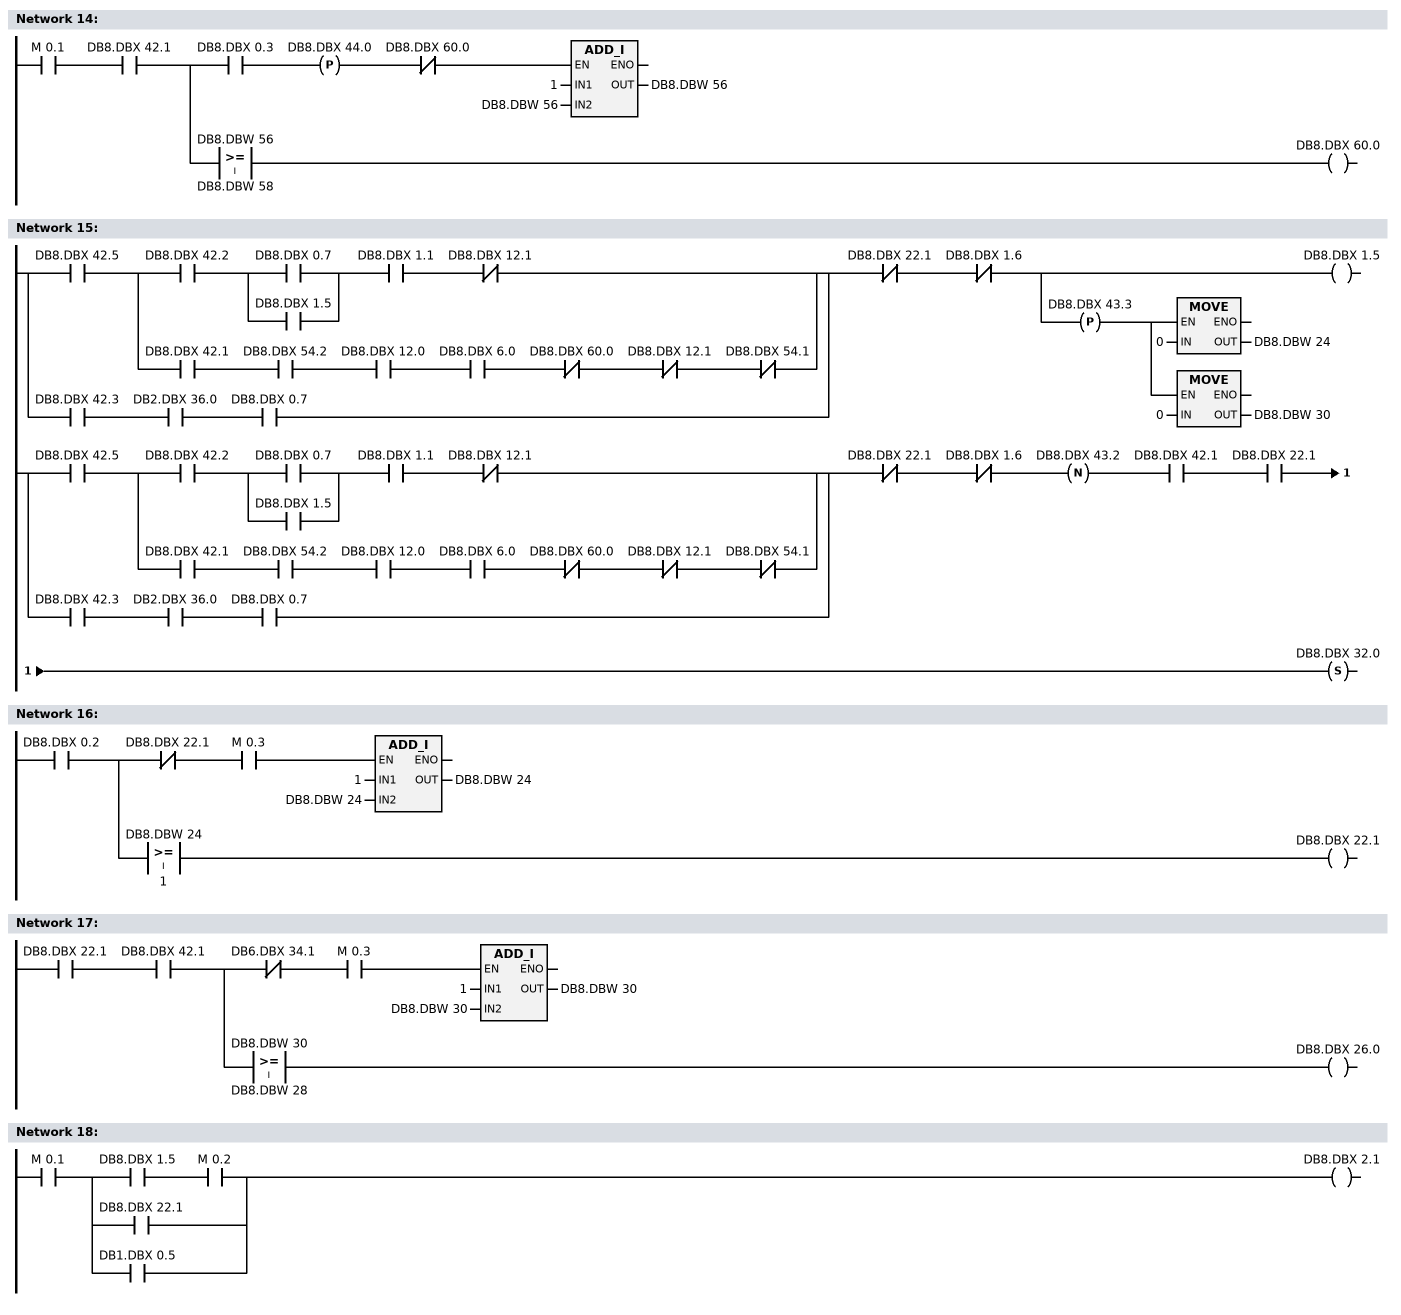
NETWORK
TITLE =
      A     M 0.1;
      A     DB8.DBX 42.1;
      =     L 0.0;
      A     L 0.0;
      A     DB8.DBX 0.3;
      FP    DB8.DBX 44.0;
      AN    DB8.DBX 60.0;
      JNB   M010;
      L     1;
      L     DB8.DBW 56;
      +I;
      T     DB8.DBW 56;
M010: NOP   0;
      A     L 0.0;
      A(;
      L     DB8.DBW 56;
      L     DB8.DBW 58;
      >=I;
      );
      =     DB8.DBX 60.0;
NETWORK
TITLE =
      A(;
      A     DB8.DBX 42.5;
      A(;
      A     DB8.DBX 42.2;
      A(;
      O     DB8.DBX 0.7;
      O     DB8.DBX 1.5;
      );
      A     DB8.DBX 1.1;
      AN    DB8.DBX 12.1;
      O;
      A     DB8.DBX 42.1;
      A     DB8.DBX 54.2;
      A     DB8.DBX 12.0;
      A     DB8.DBX 6.0;
      AN    DB8.DBX 60.0;
      AN    DB8.DBX 12.1;
      AN    DB8.DBX 54.1;
      );
      O;
      A     DB8.DBX 42.3;
      A     DB2.DBX 36.0;
      A     DB8.DBX 0.7;
      );
      AN    DB8.DBX 22.1;
      AN    DB8.DBX 1.6;
      =     L 0.0;
      A     L 0.0;
      BLD   102;
      =     DB8.DBX 1.5;
      A(;
      A     L 0.0;
      FN    DB8.DBX 43.2;
      );
      A     DB8.DBX 42.1;
      A     DB8.DBX 22.1;
      S     DB8.DBX 32.0;
      A     L 0.0;
      FP    DB8.DBX 43.3;
      =     L 0.1;
      A     L 0.1;
      JNB   M011;
      L     0;
      T     DB8.DBW 24;
M011: NOP   0;
      A     L 0.1;
      JNB   M012;
      L     0;
      T     DB8.DBW 30;
M012: NOP   0;
NETWORK
TITLE =
      A     DB8.DBX 0.2;
      =     L 0.0;
      A     L 0.0;
      AN    DB8.DBX 22.1;
      A     M 0.3;
      JNB   M013;
      L     1;
      L     DB8.DBW 24;
      +I;
      T     DB8.DBW 24;
M013: NOP   0;
      A     L 0.0;
      A(;
      L     DB8.DBW 24;
      L     1;
      >=I;
      );
      =     DB8.DBX 22.1;
NETWORK
TITLE =
      A     DB8.DBX 22.1;
      A     DB8.DBX 42.1;
      =     L 0.0;
      A     L 0.0;
      AN    DB6.DBX 34.1;
      A     M 0.3;
      JNB   M014;
      L     1;
      L     DB8.DBW 30;
      +I;
      T     DB8.DBW 30;
M014: NOP   0;
      A     L 0.0;
      A(;
      L     DB8.DBW 30;
      L     DB8.DBW 28;
      >=I;
      );
      =     DB8.DBX 26.0;
NETWORK
TITLE =
      A     M 0.1;
      A(;
      A     DB8.DBX 1.5;
      A     M 0.2;
      O     DB8.DBX 22.1;
      O     DB1.DBX 0.5;
      );
      =     DB8.DBX 2.1;
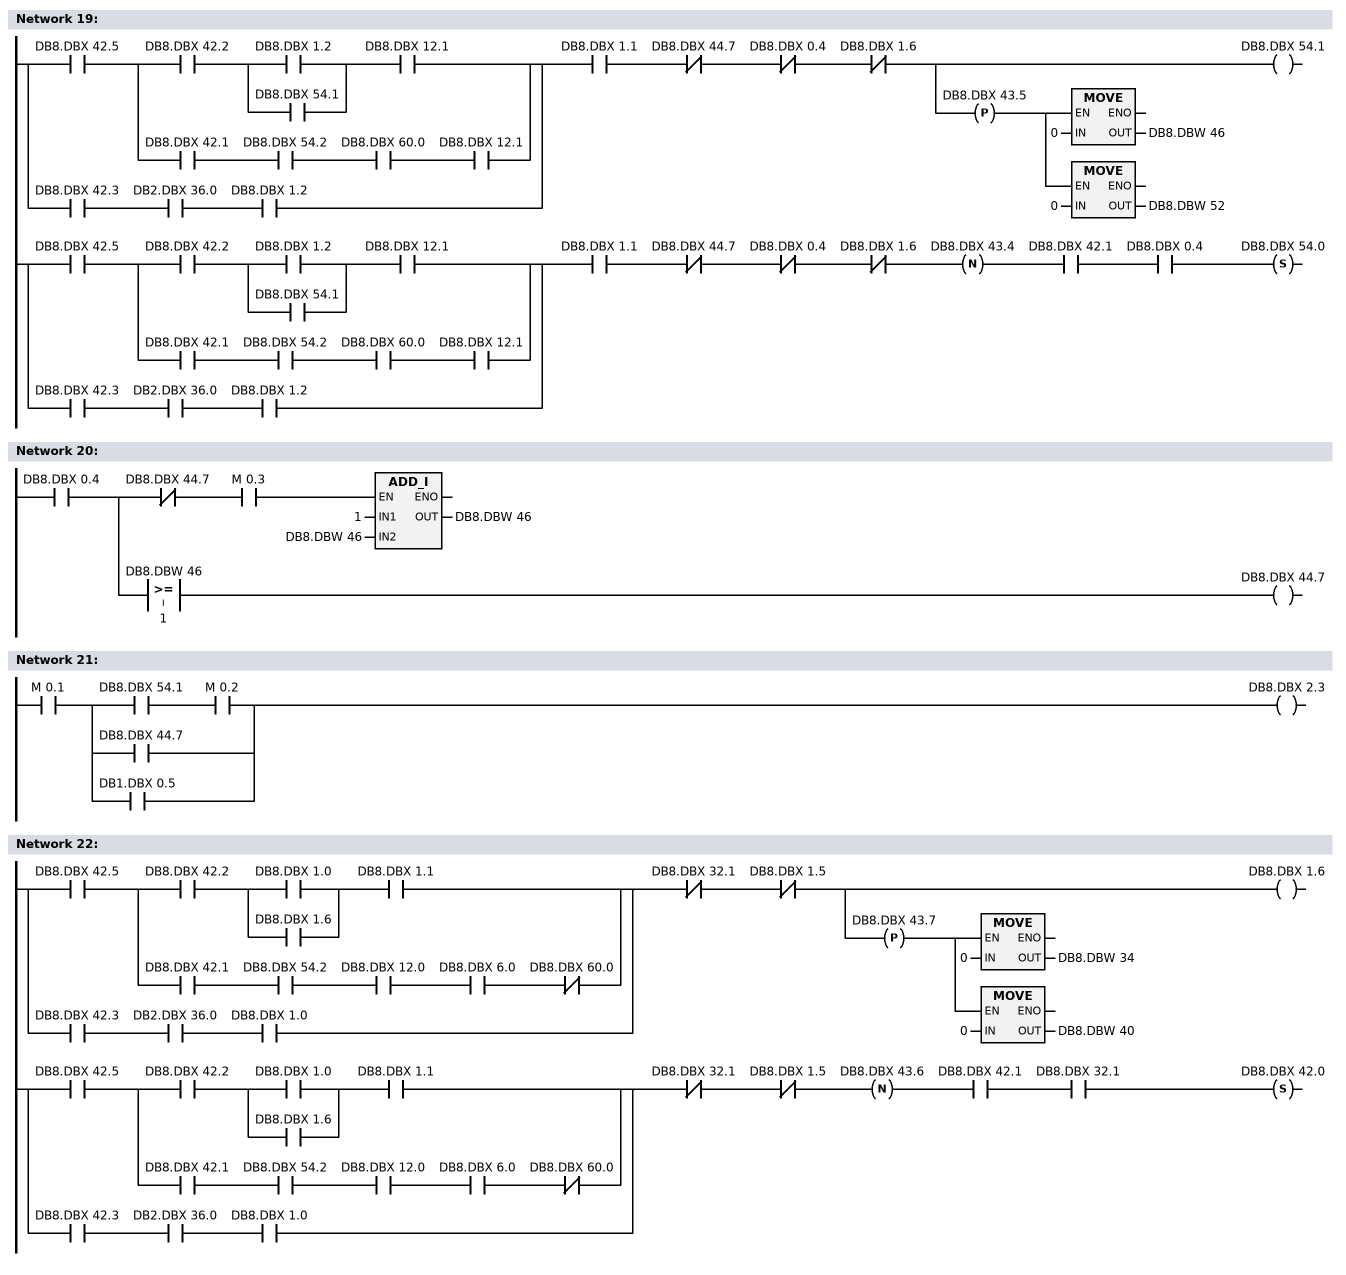
NETWORK
TITLE =
      A(;
      A     DB8.DBX 42.5;
      A(;
      A     DB8.DBX 42.2;
      A(;
      O     DB8.DBX 1.2;
      O     DB8.DBX 54.1;
      );
      A     DB8.DBX 12.1;
      O;
      A     DB8.DBX 42.1;
      A     DB8.DBX 54.2;
      A     DB8.DBX 60.0;
      A     DB8.DBX 12.1;
      );
      O;
      A     DB8.DBX 42.3;
      A     DB2.DBX 36.0;
      A     DB8.DBX 1.2;
      );
      A     DB8.DBX 1.1;
      AN    DB8.DBX 44.7;
      AN    DB8.DBX 0.4;
      AN    DB8.DBX 1.6;
      =     L 0.0;
      A     L 0.0;
      BLD   102;
      =     DB8.DBX 54.1;
      A(;
      A     L 0.0;
      FN    DB8.DBX 43.4;
      );
      A     DB8.DBX 42.1;
      A     DB8.DBX 0.4;
      S     DB8.DBX 54.0;
      A     L 0.0;
      FP    DB8.DBX 43.5;
      =     L 0.1;
      A     L 0.1;
      JNB   M015;
      L     0;
      T     DB8.DBW 46;
M015: NOP   0;
      A     L 0.1;
      JNB   M016;
      L     0;
      T     DB8.DBW 52;
M016: NOP   0;
NETWORK
TITLE =
      A     DB8.DBX 0.4;
      =     L 0.0;
      A     L 0.0;
      AN    DB8.DBX 44.7;
      A     M 0.3;
      JNB   M017;
      L     1;
      L     DB8.DBW 46;
      +I;
      T     DB8.DBW 46;
M017: NOP   0;
      A     L 0.0;
      A(;
      L     DB8.DBW 46;
      L     1;
      >=I;
      );
      =     DB8.DBX 44.7;
NETWORK
TITLE =
      A     M 0.1;
      A(;
      A     DB8.DBX 54.1;
      A     M 0.2;
      O     DB8.DBX 44.7;
      O     DB1.DBX 0.5;
      );
      =     DB8.DBX 2.3;
NETWORK
TITLE =
      A(;
      A     DB8.DBX 42.5;
      A(;
      A     DB8.DBX 42.2;
      A(;
      O     DB8.DBX 1.0;
      O     DB8.DBX 1.6;
      );
      A     DB8.DBX 1.1;
      O;
      A     DB8.DBX 42.1;
      A     DB8.DBX 54.2;
      A     DB8.DBX 12.0;
      A     DB8.DBX 6.0;
      AN    DB8.DBX 60.0;
      );
      O;
      A     DB8.DBX 42.3;
      A     DB2.DBX 36.0;
      A     DB8.DBX 1.0;
      );
      AN    DB8.DBX 32.1;
      AN    DB8.DBX 1.5;
      =     L 0.0;
      A     L 0.0;
      BLD   102;
      =     DB8.DBX 1.6;
      A(;
      A     L 0.0;
      FN    DB8.DBX 43.6;
      );
      A     DB8.DBX 42.1;
      A     DB8.DBX 32.1;
      S     DB8.DBX 42.0;
      A     L 0.0;
      FP    DB8.DBX 43.7;
      =     L 0.1;
      A     L 0.1;
      JNB   M018;
      L     0;
      T     DB8.DBW 34;
M018: NOP   0;
      A     L 0.1;
      JNB   M019;
      L     0;
      T     DB8.DBW 40;
M019: NOP   0;
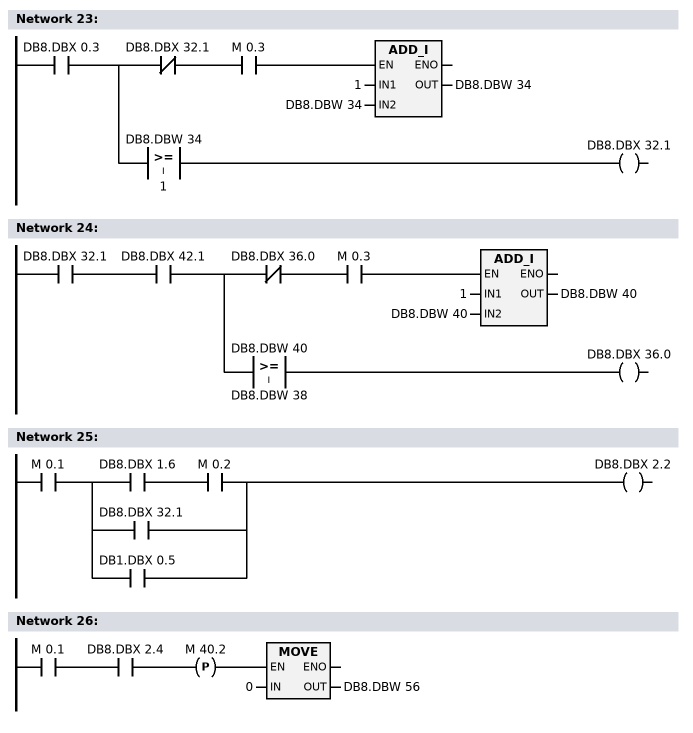
NETWORK
TITLE =
      A     DB8.DBX 0.3;
      =     L 0.0;
      A     L 0.0;
      AN    DB8.DBX 32.1;
      A     M 0.3;
      JNB   M020;
      L     1;
      L     DB8.DBW 34;
      +I;
      T     DB8.DBW 34;
M020: NOP   0;
      A     L 0.0;
      A(;
      L     DB8.DBW 34;
      L     1;
      >=I;
      );
      =     DB8.DBX 32.1;
NETWORK
TITLE =
      A     DB8.DBX 32.1;
      A     DB8.DBX 42.1;
      =     L 0.0;
      A     L 0.0;
      AN    DB8.DBX 36.0;
      A     M 0.3;
      JNB   M021;
      L     1;
      L     DB8.DBW 40;
      +I;
      T     DB8.DBW 40;
M021: NOP   0;
      A     L 0.0;
      A(;
      L     DB8.DBW 40;
      L     DB8.DBW 38;
      >=I;
      );
      =     DB8.DBX 36.0;
NETWORK
TITLE =
      A     M 0.1;
      A(;
      A     DB8.DBX 1.6;
      A     M 0.2;
      O     DB8.DBX 32.1;
      O     DB1.DBX 0.5;
      );
      =     DB8.DBX 2.2;
NETWORK
TITLE =
      A     M 0.1;
      A     DB8.DBX 2.4;
      FP    M 40.2;
      JNB   M022;
      L     0;
      T     DB8.DBW 56;
M022: NOP   0;
END_FUNCTION

FUNCTION FC 11 : VOID
AUTHOR : Kamillas
VERSION : 0.1
BEGIN
// (block stored without names or comments; labels and parameter names are numbered)
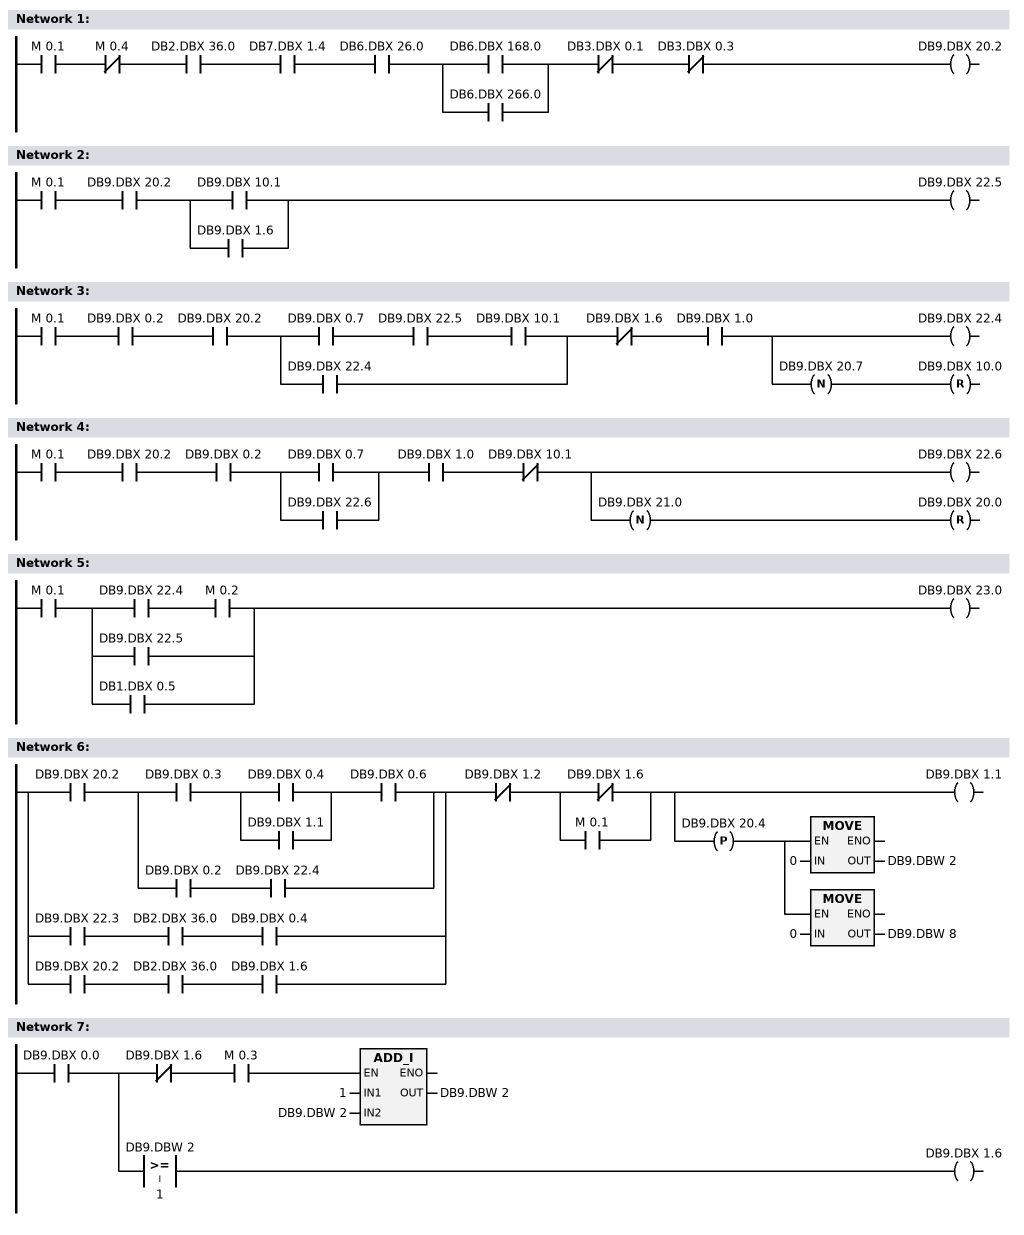
NETWORK
TITLE =
      A     M 0.1;
      AN    M 0.4;
      A     DB2.DBX 36.0;
      A     DB7.DBX 1.4;
      A     DB6.DBX 26.0;
      A(;
      O     DB6.DBX 168.0;
      O     DB6.DBX 266.0;
      );
      AN    DB3.DBX 0.1;
      AN    DB3.DBX 0.3;
      =     DB9.DBX 20.2;
NETWORK
TITLE =
      A     M 0.1;
      A     DB9.DBX 20.2;
      A(;
      O     DB9.DBX 10.1;
      O     DB9.DBX 1.6;
      );
      =     DB9.DBX 22.5;
NETWORK
TITLE =
      A     M 0.1;
      A     DB9.DBX 0.2;
      A     DB9.DBX 20.2;
      A(;
      A     DB9.DBX 0.7;
      A     DB9.DBX 22.5;
      A     DB9.DBX 10.1;
      O     DB9.DBX 22.4;
      );
      AN    DB9.DBX 1.6;
      A     DB9.DBX 1.0;
      =     L 0.0;
      A     L 0.0;
      BLD   102;
      =     DB9.DBX 22.4;
      A     L 0.0;
      FN    DB9.DBX 20.7;
      R     DB9.DBX 10.0;
NETWORK
TITLE =
      A     M 0.1;
      A     DB9.DBX 20.2;
      A     DB9.DBX 0.2;
      A(;
      O     DB9.DBX 0.7;
      O     DB9.DBX 22.6;
      );
      A     DB9.DBX 1.0;
      AN    DB9.DBX 10.1;
      =     L 0.0;
      A     L 0.0;
      BLD   102;
      =     DB9.DBX 22.6;
      A     L 0.0;
      FN    DB9.DBX 21.0;
      R     DB9.DBX 20.0;
NETWORK
TITLE =
      A     M 0.1;
      A(;
      A     DB9.DBX 22.4;
      A     M 0.2;
      O     DB9.DBX 22.5;
      O     DB1.DBX 0.5;
      );
      =     DB9.DBX 23.0;
NETWORK
TITLE =
      A(;
      A     DB9.DBX 20.2;
      A(;
      A     DB9.DBX 0.3;
      A(;
      O     DB9.DBX 0.4;
      O     DB9.DBX 1.1;
      );
      A     DB9.DBX 0.6;
      O;
      A     DB9.DBX 0.2;
      A     DB9.DBX 22.4;
      );
      O;
      A     DB9.DBX 22.3;
      A     DB2.DBX 36.0;
      A     DB9.DBX 0.4;
      O;
      A     DB9.DBX 20.2;
      A     DB2.DBX 36.0;
      A     DB9.DBX 1.6;
      );
      AN    DB9.DBX 1.2;
      A(;
      ON    DB9.DBX 1.6;
      O     M 0.1;
      );
      =     L 0.0;
      A     L 0.0;
      BLD   102;
      =     DB9.DBX 1.1;
      A     L 0.0;
      FP    DB9.DBX 20.4;
      =     L 0.1;
      A     L 0.1;
      JNB   M001;
      L     0;
      T     DB9.DBW 2;
M001: NOP   0;
      A     L 0.1;
      JNB   M002;
      L     0;
      T     DB9.DBW 8;
M002: NOP   0;
NETWORK
TITLE =
      A     DB9.DBX 0.0;
      =     L 0.0;
      A     L 0.0;
      AN    DB9.DBX 1.6;
      A     M 0.3;
      JNB   M003;
      L     1;
      L     DB9.DBW 2;
      +I;
      T     DB9.DBW 2;
M003: NOP   0;
      A     L 0.0;
      A(;
      L     DB9.DBW 2;
      L     1;
      >=I;
      );
      =     DB9.DBX 1.6;
NETWORK
TITLE =
      A     DB9.DBX 1.6;
      =     L 0.0;
      A     L 0.0;
      A     DB9.DBX 0.2;
      AN    DB9.DBX 4.0;
      A     M 0.3;
      JNB   M004;
      L     1;
      L     DB9.DBW 8;
      +I;
      T     DB9.DBW 8;
M004: NOP   0;
      A     L 0.0;
      A(;
      L     DB9.DBW 8;
      L     DB9.DBW 6;
      >=I;
      );
      =     L 0.1;
      A     L 0.1;
      A     DB9.DBX 0.2;
      =     DB9.DBX 4.0;
      A(;
      A     L 0.1;
      FP    DB9.DBX 20.3;
      );
      A     DB9.DBX 0.2;
      A     DB9.DBX 1.6;
      S     DB9.DBX 10.0;
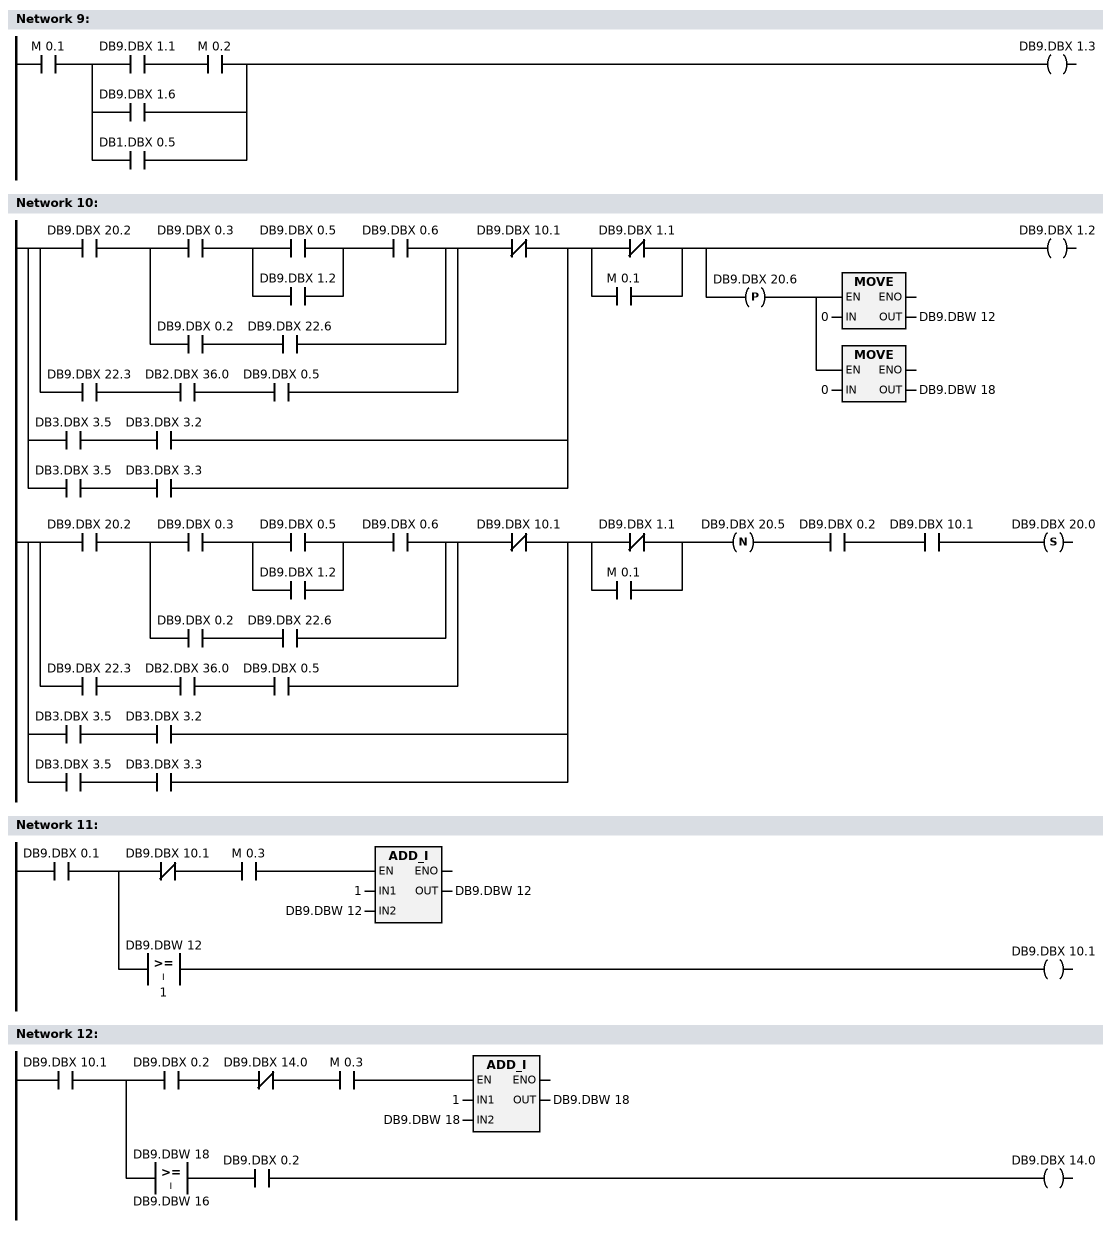
NETWORK
TITLE =
      A     M 0.1;
      A(;
      A     DB9.DBX 1.1;
      A     M 0.2;
      O     DB9.DBX 1.6;
      O     DB1.DBX 0.5;
      );
      =     DB9.DBX 1.3;
NETWORK
TITLE =
      A(;
      A(;
      A     DB9.DBX 20.2;
      A(;
      A     DB9.DBX 0.3;
      A(;
      O     DB9.DBX 0.5;
      O     DB9.DBX 1.2;
      );
      A     DB9.DBX 0.6;
      O;
      A     DB9.DBX 0.2;
      A     DB9.DBX 22.6;
      );
      O;
      A     DB9.DBX 22.3;
      A     DB2.DBX 36.0;
      A     DB9.DBX 0.5;
      );
      AN    DB9.DBX 10.1;
      O;
      A     DB3.DBX 3.5;
      A     DB3.DBX 3.2;
      O;
      A     DB3.DBX 3.5;
      A     DB3.DBX 3.3;
      );
      A(;
      ON    DB9.DBX 1.1;
      O     M 0.1;
      );
      =     L 0.0;
      A     L 0.0;
      BLD   102;
      =     DB9.DBX 1.2;
      A(;
      A     L 0.0;
      FN    DB9.DBX 20.5;
      );
      A     DB9.DBX 0.2;
      A     DB9.DBX 10.1;
      S     DB9.DBX 20.0;
      A     L 0.0;
      FP    DB9.DBX 20.6;
      =     L 0.1;
      A     L 0.1;
      JNB   M005;
      L     0;
      T     DB9.DBW 12;
M005: NOP   0;
      A     L 0.1;
      JNB   M006;
      L     0;
      T     DB9.DBW 18;
M006: NOP   0;
NETWORK
TITLE =
      A     DB9.DBX 0.1;
      =     L 0.0;
      A     L 0.0;
      AN    DB9.DBX 10.1;
      A     M 0.3;
      JNB   M007;
      L     1;
      L     DB9.DBW 12;
      +I;
      T     DB9.DBW 12;
M007: NOP   0;
      A     L 0.0;
      A(;
      L     DB9.DBW 12;
      L     1;
      >=I;
      );
      =     DB9.DBX 10.1;
NETWORK
TITLE =
      A     DB9.DBX 10.1;
      =     L 0.0;
      A     L 0.0;
      A     DB9.DBX 0.2;
      AN    DB9.DBX 14.0;
      A     M 0.3;
      JNB   M008;
      L     1;
      L     DB9.DBW 18;
      +I;
      T     DB9.DBW 18;
M008: NOP   0;
      A     L 0.0;
      A(;
      L     DB9.DBW 18;
      L     DB9.DBW 16;
      >=I;
      );
      A     DB9.DBX 0.2;
      =     DB9.DBX 14.0;
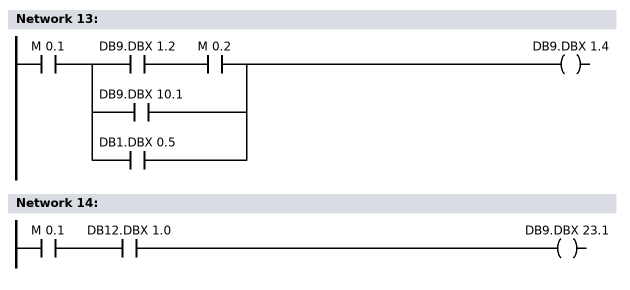
NETWORK
TITLE =
      A     M 0.1;
      A(;
      A     DB9.DBX 1.2;
      A     M 0.2;
      O     DB9.DBX 10.1;
      O     DB1.DBX 0.5;
      );
      =     DB9.DBX 1.4;
NETWORK
TITLE =
      A     M 0.1;
      A     DB12.DBX 1.0;
      =     DB9.DBX 23.1;
END_FUNCTION

FUNCTION FC 12 : VOID
AUTHOR : Kamillas
VERSION : 0.1
BEGIN
// (block stored without names or comments; labels and parameter names are numbered)
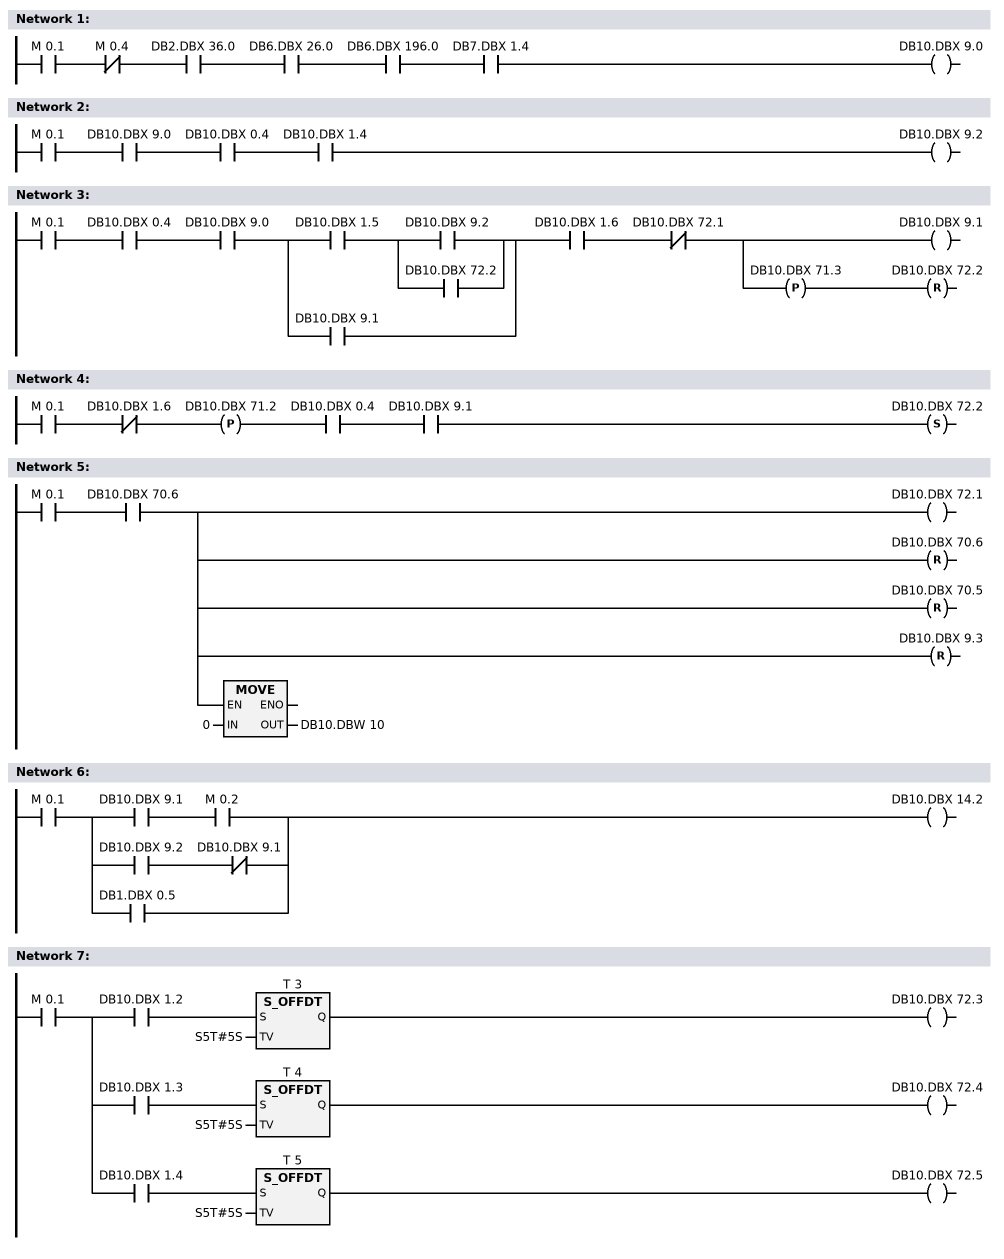
NETWORK
TITLE =
      A     M 0.1;
      AN    M 0.4;
      A     DB2.DBX 36.0;
      A     DB6.DBX 26.0;
      A     DB6.DBX 196.0;
      A     DB7.DBX 1.4;
      =     DB10.DBX 9.0;
NETWORK
TITLE =
      A     M 0.1;
      A     DB10.DBX 9.0;
      A     DB10.DBX 0.4;
      A     DB10.DBX 1.4;
      =     DB10.DBX 9.2;
NETWORK
TITLE =
      A     M 0.1;
      A     DB10.DBX 0.4;
      A     DB10.DBX 9.0;
      A(;
      A     DB10.DBX 1.5;
      A(;
      O     DB10.DBX 9.2;
      O     DB10.DBX 72.2;
      );
      O     DB10.DBX 9.1;
      );
      A     DB10.DBX 1.6;
      AN    DB10.DBX 72.1;
      =     L 0.0;
      A     L 0.0;
      BLD   102;
      =     DB10.DBX 9.1;
      A     L 0.0;
      FP    DB10.DBX 71.3;
      R     DB10.DBX 72.2;
NETWORK
TITLE =
      A     M 0.1;
      AN    DB10.DBX 1.6;
      FP    DB10.DBX 71.2;
      A     DB10.DBX 0.4;
      A     DB10.DBX 9.1;
      S     DB10.DBX 72.2;
NETWORK
TITLE =
      A     M 0.1;
      A     DB10.DBX 70.6;
      =     L 0.0;
      A     L 0.0;
      BLD   102;
      =     DB10.DBX 72.1;
      A     L 0.0;
      BLD   102;
      R     DB10.DBX 70.6;
      A     L 0.0;
      BLD   102;
      R     DB10.DBX 70.5;
      A     L 0.0;
      BLD   102;
      R     DB10.DBX 9.3;
      A     L 0.0;
      JNB   M001;
      L     0;
      T     DB10.DBW 10;
M001: NOP   0;
NETWORK
TITLE =
      A     M 0.1;
      A(;
      A     DB10.DBX 9.1;
      A     M 0.2;
      O;
      A     DB10.DBX 9.2;
      AN    DB10.DBX 9.1;
      O     DB1.DBX 0.5;
      );
      =     DB10.DBX 14.2;
NETWORK
TITLE =
      A     M 0.1;
      =     L 0.0;
      A     L 0.0;
      A     DB10.DBX 1.2;
      L     S5T#5S;
      SF    T 3;
      NOP   0;
      NOP   0;
      NOP   0;
      A     T 3;
      =     DB10.DBX 72.3;
      A     L 0.0;
      A     DB10.DBX 1.3;
      L     S5T#5S;
      SF    T 4;
      NOP   0;
      NOP   0;
      NOP   0;
      A     T 4;
      =     DB10.DBX 72.4;
      A     L 0.0;
      A     DB10.DBX 1.4;
      L     S5T#5S;
      SF    T 5;
      NOP   0;
      NOP   0;
      NOP   0;
      A     T 5;
      =     DB10.DBX 72.5;
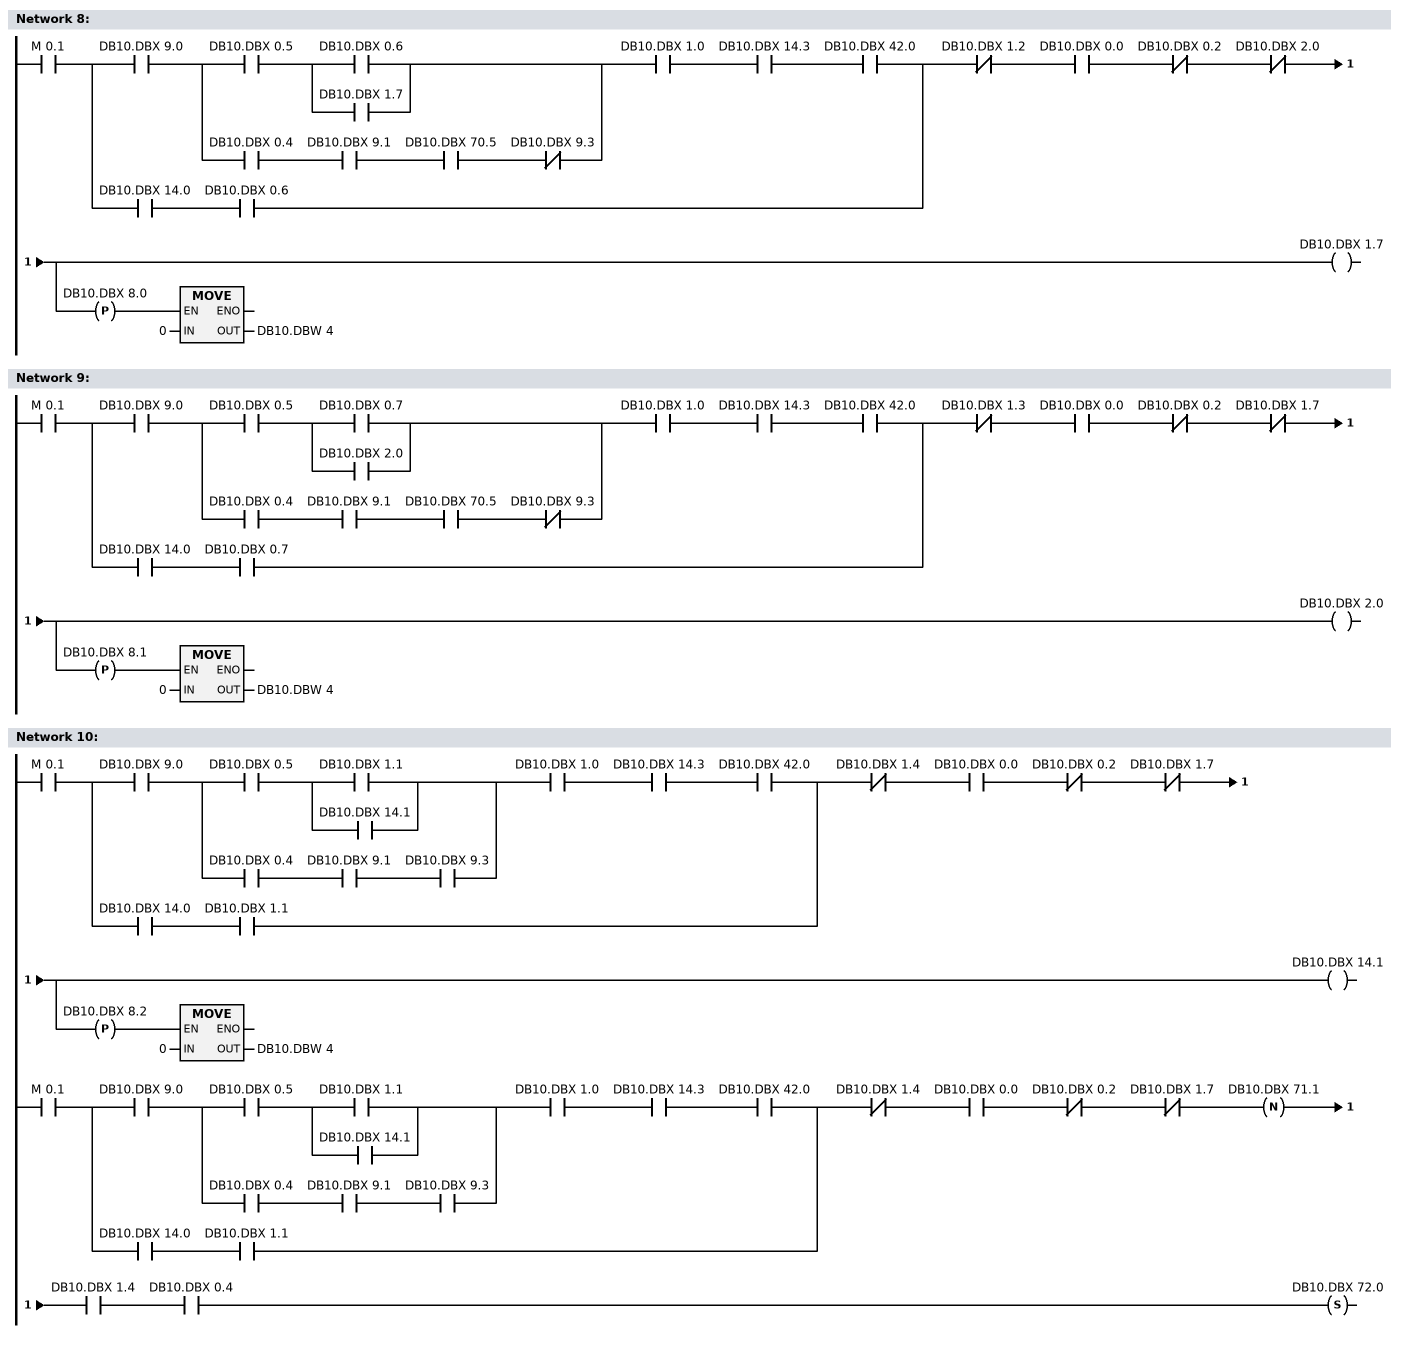
NETWORK
TITLE =
      A     M 0.1;
      A(;
      A     DB10.DBX 9.0;
      A(;
      A     DB10.DBX 0.5;
      A(;
      O     DB10.DBX 0.6;
      O     DB10.DBX 1.7;
      );
      O;
      A     DB10.DBX 0.4;
      A     DB10.DBX 9.1;
      A     DB10.DBX 70.5;
      AN    DB10.DBX 9.3;
      );
      A     DB10.DBX 1.0;
      A     DB10.DBX 14.3;
      A     DB10.DBX 42.0;
      O;
      A     DB10.DBX 14.0;
      A     DB10.DBX 0.6;
      );
      AN    DB10.DBX 1.2;
      A     DB10.DBX 0.0;
      AN    DB10.DBX 0.2;
      AN    DB10.DBX 2.0;
      =     L 0.0;
      A     L 0.0;
      BLD   102;
      =     DB10.DBX 1.7;
      A     L 0.0;
      FP    DB10.DBX 8.0;
      JNB   M002;
      L     0;
      T     DB10.DBW 4;
M002: NOP   0;
NETWORK
TITLE =
      A     M 0.1;
      A(;
      A     DB10.DBX 9.0;
      A(;
      A     DB10.DBX 0.5;
      A(;
      O     DB10.DBX 0.7;
      O     DB10.DBX 2.0;
      );
      O;
      A     DB10.DBX 0.4;
      A     DB10.DBX 9.1;
      A     DB10.DBX 70.5;
      AN    DB10.DBX 9.3;
      );
      A     DB10.DBX 1.0;
      A     DB10.DBX 14.3;
      A     DB10.DBX 42.0;
      O;
      A     DB10.DBX 14.0;
      A     DB10.DBX 0.7;
      );
      AN    DB10.DBX 1.3;
      A     DB10.DBX 0.0;
      AN    DB10.DBX 0.2;
      AN    DB10.DBX 1.7;
      =     L 0.0;
      A     L 0.0;
      BLD   102;
      =     DB10.DBX 2.0;
      A     L 0.0;
      FP    DB10.DBX 8.1;
      JNB   M003;
      L     0;
      T     DB10.DBW 4;
M003: NOP   0;
NETWORK
TITLE =
      A     M 0.1;
      A(;
      A     DB10.DBX 9.0;
      A(;
      A     DB10.DBX 0.5;
      A(;
      O     DB10.DBX 1.1;
      O     DB10.DBX 14.1;
      );
      O;
      A     DB10.DBX 0.4;
      A     DB10.DBX 9.1;
      A     DB10.DBX 9.3;
      );
      A     DB10.DBX 1.0;
      A     DB10.DBX 14.3;
      A     DB10.DBX 42.0;
      O;
      A     DB10.DBX 14.0;
      A     DB10.DBX 1.1;
      );
      AN    DB10.DBX 1.4;
      A     DB10.DBX 0.0;
      AN    DB10.DBX 0.2;
      AN    DB10.DBX 1.7;
      =     L 0.0;
      A     L 0.0;
      BLD   102;
      =     DB10.DBX 14.1;
      A(;
      A     L 0.0;
      FN    DB10.DBX 71.1;
      );
      A     DB10.DBX 1.4;
      A     DB10.DBX 0.4;
      S     DB10.DBX 72.0;
      A     L 0.0;
      FP    DB10.DBX 8.2;
      JNB   M004;
      L     0;
      T     DB10.DBW 4;
M004: NOP   0;
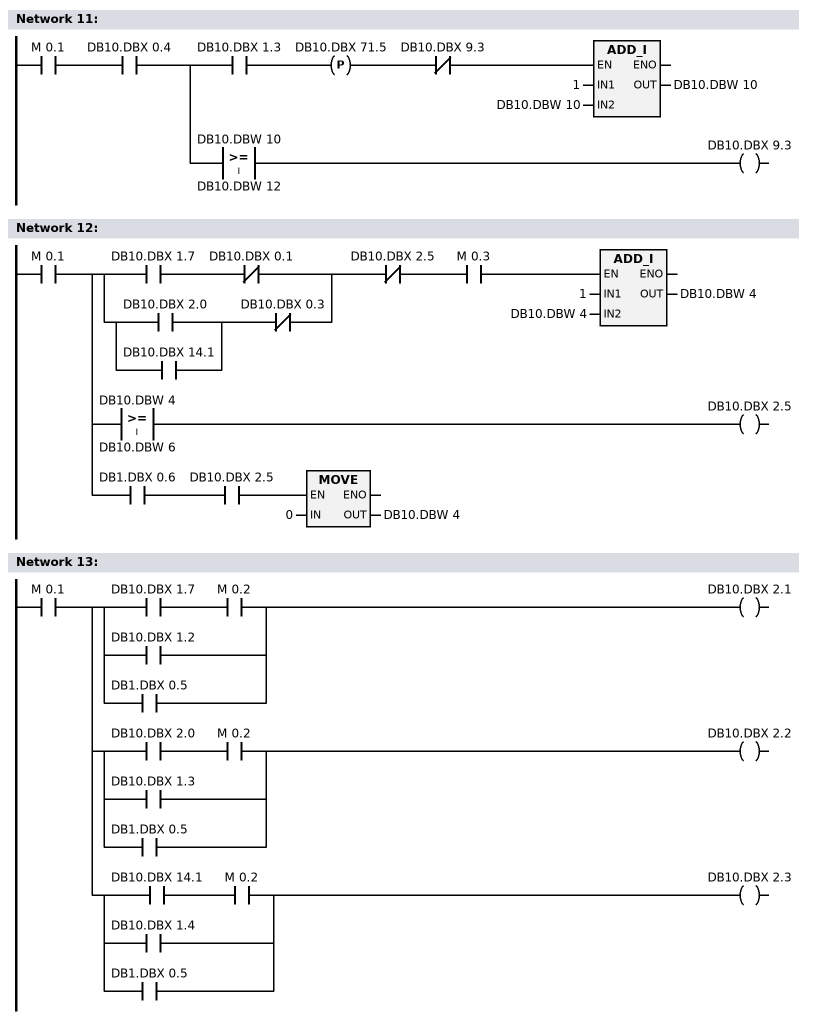
NETWORK
TITLE =
      A     M 0.1;
      A     DB10.DBX 0.4;
      =     L 0.0;
      A     L 0.0;
      A     DB10.DBX 1.3;
      FP    DB10.DBX 71.5;
      AN    DB10.DBX 9.3;
      JNB   M005;
      L     1;
      L     DB10.DBW 10;
      +I;
      T     DB10.DBW 10;
M005: NOP   0;
      A     L 0.0;
      A(;
      L     DB10.DBW 10;
      L     DB10.DBW 12;
      >=I;
      );
      =     DB10.DBX 9.3;
NETWORK
TITLE =
      A     M 0.1;
      =     L 0.0;
      A     L 0.0;
      A(;
      A     DB10.DBX 1.7;
      AN    DB10.DBX 0.1;
      O;
      A(;
      O     DB10.DBX 2.0;
      O     DB10.DBX 14.1;
      );
      AN    DB10.DBX 0.3;
      );
      AN    DB10.DBX 2.5;
      A     M 0.3;
      JNB   M006;
      L     1;
      L     DB10.DBW 4;
      +I;
      T     DB10.DBW 4;
M006: NOP   0;
      A     L 0.0;
      A(;
      L     DB10.DBW 4;
      L     DB10.DBW 6;
      >=I;
      );
      =     DB10.DBX 2.5;
      A     L 0.0;
      A     DB1.DBX 0.6;
      A     DB10.DBX 2.5;
      JNB   M007;
      L     0;
      T     DB10.DBW 4;
M007: NOP   0;
NETWORK
TITLE =
      A     M 0.1;
      =     L 0.0;
      A     L 0.0;
      A(;
      A     DB10.DBX 1.7;
      A     M 0.2;
      O     DB10.DBX 1.2;
      O     DB1.DBX 0.5;
      );
      =     DB10.DBX 2.1;
      A     L 0.0;
      A(;
      A     DB10.DBX 2.0;
      A     M 0.2;
      O     DB10.DBX 1.3;
      O     DB1.DBX 0.5;
      );
      =     DB10.DBX 2.2;
      A     L 0.0;
      A(;
      A     DB10.DBX 14.1;
      A     M 0.2;
      O     DB10.DBX 1.4;
      O     DB1.DBX 0.5;
      );
      =     DB10.DBX 2.3;
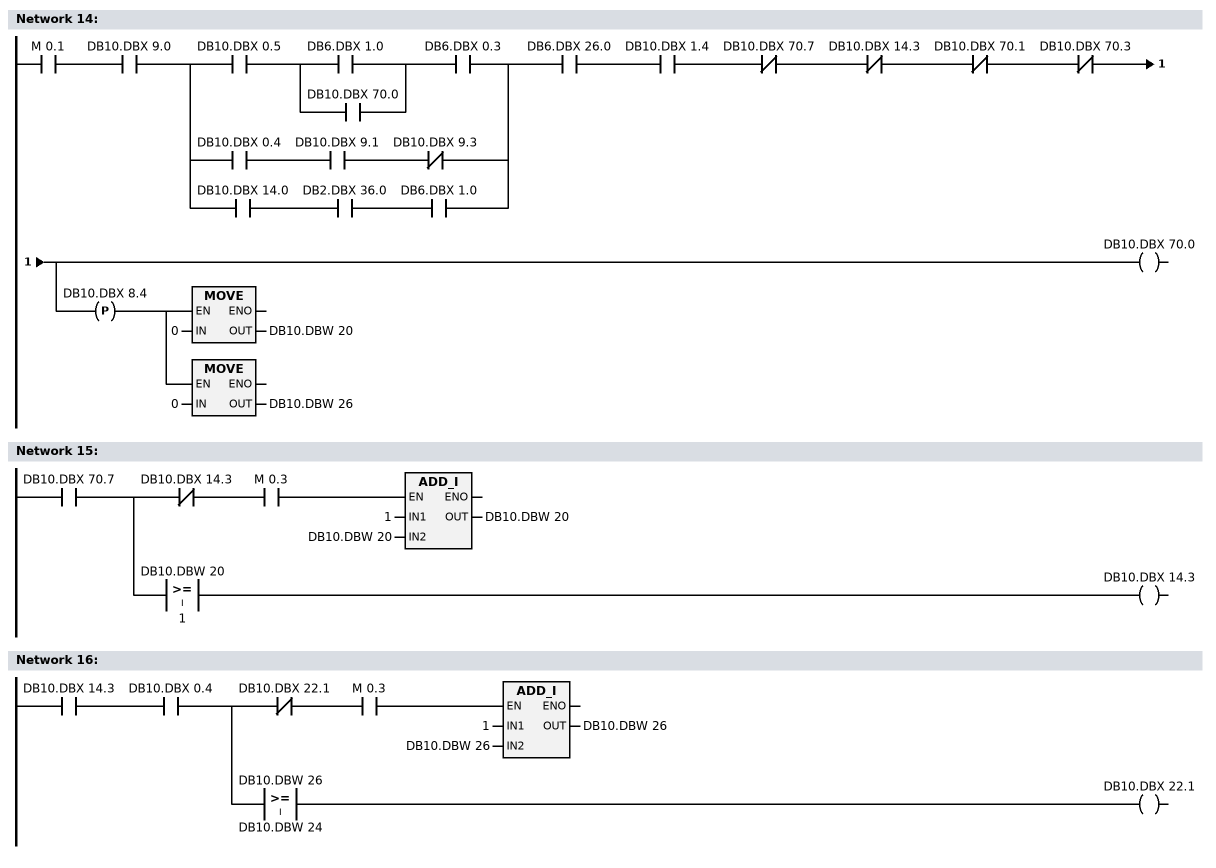
NETWORK
TITLE =
      A     M 0.1;
      A     DB10.DBX 9.0;
      A(;
      A     DB10.DBX 0.5;
      A(;
      O     DB6.DBX 1.0;
      O     DB10.DBX 70.0;
      );
      A     DB6.DBX 0.3;
      O;
      A     DB10.DBX 0.4;
      A     DB10.DBX 9.1;
      AN    DB10.DBX 9.3;
      O;
      A     DB10.DBX 14.0;
      A     DB2.DBX 36.0;
      A     DB6.DBX 1.0;
      );
      A     DB6.DBX 26.0;
      A     DB10.DBX 1.4;
      AN    DB10.DBX 70.7;
      AN    DB10.DBX 14.3;
      AN    DB10.DBX 70.1;
      AN    DB10.DBX 70.3;
      =     L 0.0;
      A     L 0.0;
      BLD   102;
      =     DB10.DBX 70.0;
      A     L 0.0;
      FP    DB10.DBX 8.4;
      =     L 0.1;
      A     L 0.1;
      JNB   M008;
      L     0;
      T     DB10.DBW 20;
M008: NOP   0;
      A     L 0.1;
      JNB   M009;
      L     0;
      T     DB10.DBW 26;
M009: NOP   0;
NETWORK
TITLE =
      A     DB10.DBX 70.7;
      =     L 0.0;
      A     L 0.0;
      AN    DB10.DBX 14.3;
      A     M 0.3;
      JNB   M010;
      L     1;
      L     DB10.DBW 20;
      +I;
      T     DB10.DBW 20;
M010: NOP   0;
      A     L 0.0;
      A(;
      L     DB10.DBW 20;
      L     1;
      >=I;
      );
      =     DB10.DBX 14.3;
NETWORK
TITLE =
      A     DB10.DBX 14.3;
      A     DB10.DBX 0.4;
      =     L 0.0;
      A     L 0.0;
      AN    DB10.DBX 22.1;
      A     M 0.3;
      JNB   M011;
      L     1;
      L     DB10.DBW 26;
      +I;
      T     DB10.DBW 26;
M011: NOP   0;
      A     L 0.0;
      A(;
      L     DB10.DBW 26;
      L     DB10.DBW 24;
      >=I;
      );
      =     DB10.DBX 22.1;
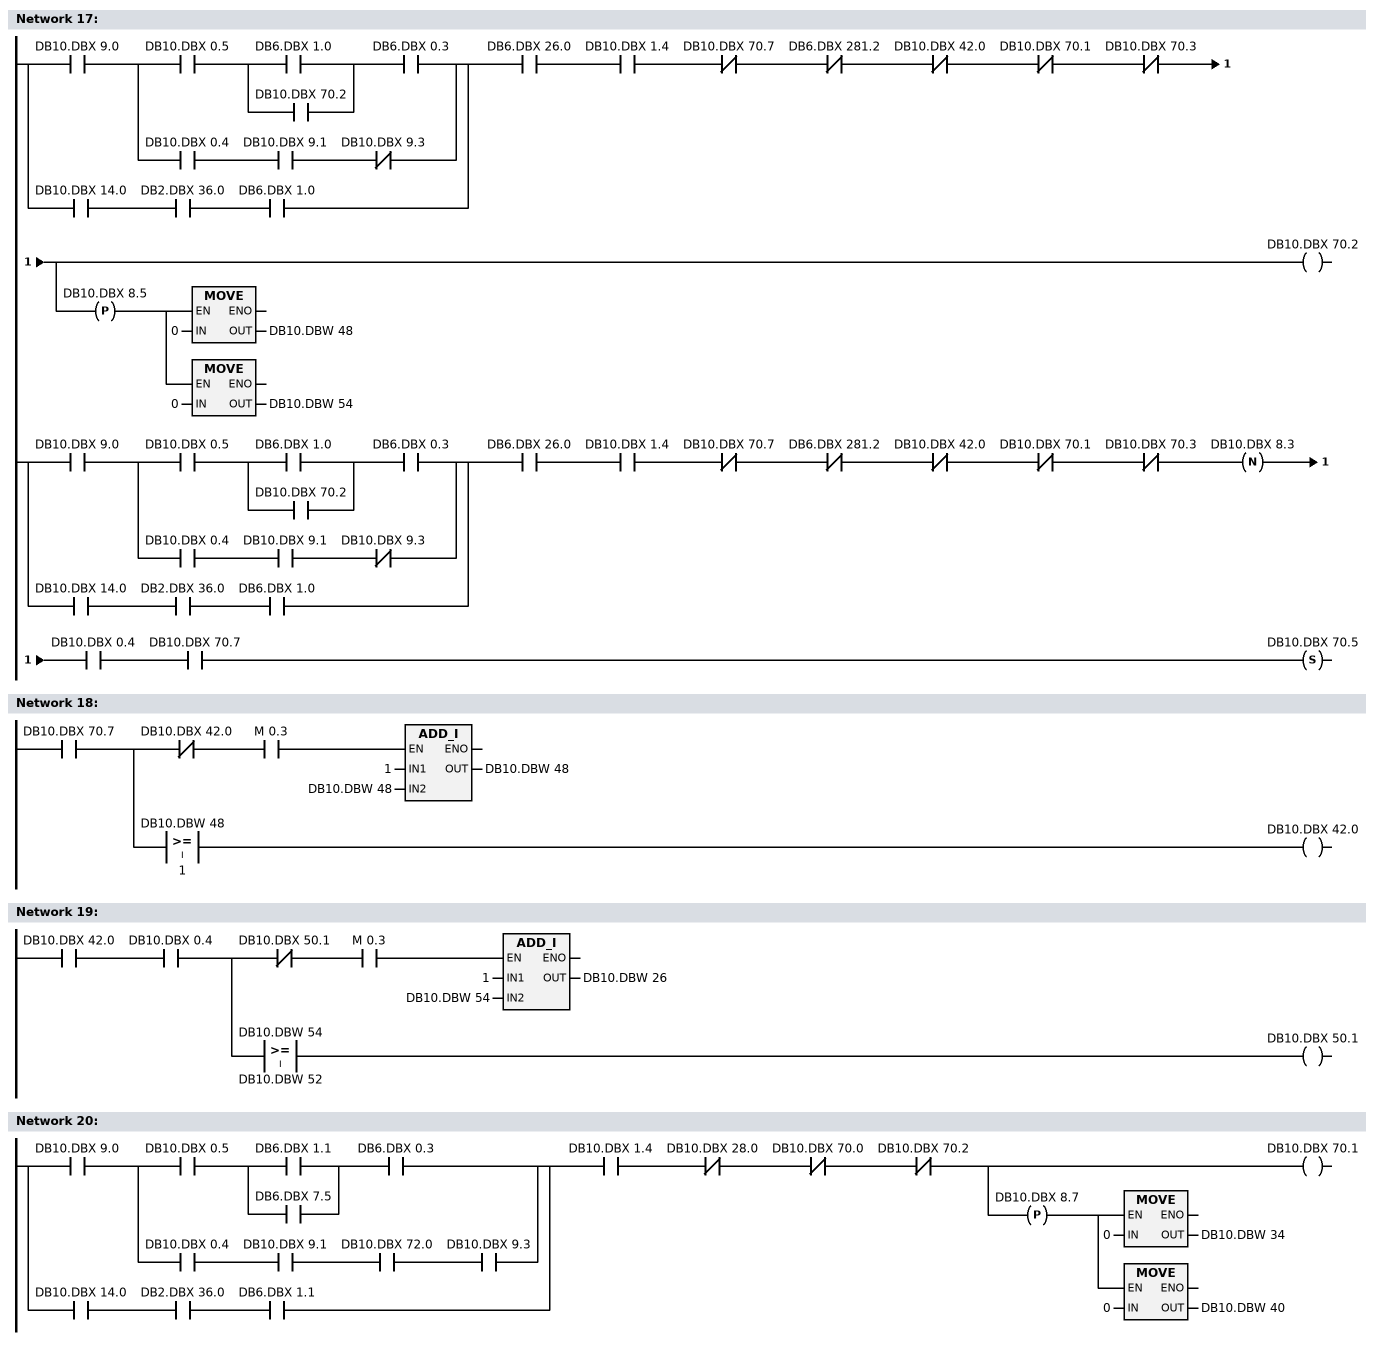
NETWORK
TITLE =
      A(;
      A     DB10.DBX 9.0;
      A(;
      A     DB10.DBX 0.5;
      A(;
      O     DB6.DBX 1.0;
      O     DB10.DBX 70.2;
      );
      A     DB6.DBX 0.3;
      O;
      A     DB10.DBX 0.4;
      A     DB10.DBX 9.1;
      AN    DB10.DBX 9.3;
      );
      O;
      A     DB10.DBX 14.0;
      A     DB2.DBX 36.0;
      A     DB6.DBX 1.0;
      );
      A     DB6.DBX 26.0;
      A     DB10.DBX 1.4;
      AN    DB10.DBX 70.7;
      AN    DB6.DBX 281.2;
      AN    DB10.DBX 42.0;
      AN    DB10.DBX 70.1;
      AN    DB10.DBX 70.3;
      =     L 0.0;
      A     L 0.0;
      BLD   102;
      =     DB10.DBX 70.2;
      A(;
      A     L 0.0;
      FN    DB10.DBX 8.3;
      );
      A     DB10.DBX 0.4;
      A     DB10.DBX 70.7;
      S     DB10.DBX 70.5;
      A     L 0.0;
      FP    DB10.DBX 8.5;
      =     L 0.1;
      A     L 0.1;
      JNB   M012;
      L     0;
      T     DB10.DBW 48;
M012: NOP   0;
      A     L 0.1;
      JNB   M013;
      L     0;
      T     DB10.DBW 54;
M013: NOP   0;
NETWORK
TITLE =
      A     DB10.DBX 70.7;
      =     L 0.0;
      A     L 0.0;
      AN    DB10.DBX 42.0;
      A     M 0.3;
      JNB   M014;
      L     1;
      L     DB10.DBW 48;
      +I;
      T     DB10.DBW 48;
M014: NOP   0;
      A     L 0.0;
      A(;
      L     DB10.DBW 48;
      L     1;
      >=I;
      );
      =     DB10.DBX 42.0;
NETWORK
TITLE =
      A     DB10.DBX 42.0;
      A     DB10.DBX 0.4;
      =     L 0.0;
      A     L 0.0;
      AN    DB10.DBX 50.1;
      A     M 0.3;
      JNB   M015;
      L     1;
      L     DB10.DBW 54;
      +I;
      T     DB10.DBW 26;
M015: NOP   0;
      A     L 0.0;
      A(;
      L     DB10.DBW 54;
      L     DB10.DBW 52;
      >=I;
      );
      =     DB10.DBX 50.1;
NETWORK
TITLE =
      A(;
      A     DB10.DBX 9.0;
      A(;
      A     DB10.DBX 0.5;
      A(;
      O     DB6.DBX 1.1;
      O     DB6.DBX 7.5;
      );
      A     DB6.DBX 0.3;
      O;
      A     DB10.DBX 0.4;
      A     DB10.DBX 9.1;
      A     DB10.DBX 72.0;
      A     DB10.DBX 9.3;
      );
      O;
      A     DB10.DBX 14.0;
      A     DB2.DBX 36.0;
      A     DB6.DBX 1.1;
      );
      A     DB10.DBX 1.4;
      AN    DB10.DBX 28.0;
      AN    DB10.DBX 70.0;
      AN    DB10.DBX 70.2;
      =     L 0.0;
      A     L 0.0;
      BLD   102;
      =     DB10.DBX 70.1;
      A     L 0.0;
      FP    DB10.DBX 8.7;
      =     L 0.1;
      A     L 0.1;
      JNB   M016;
      L     0;
      T     DB10.DBW 34;
M016: NOP   0;
      A     L 0.1;
      JNB   M017;
      L     0;
      T     DB10.DBW 40;
M017: NOP   0;
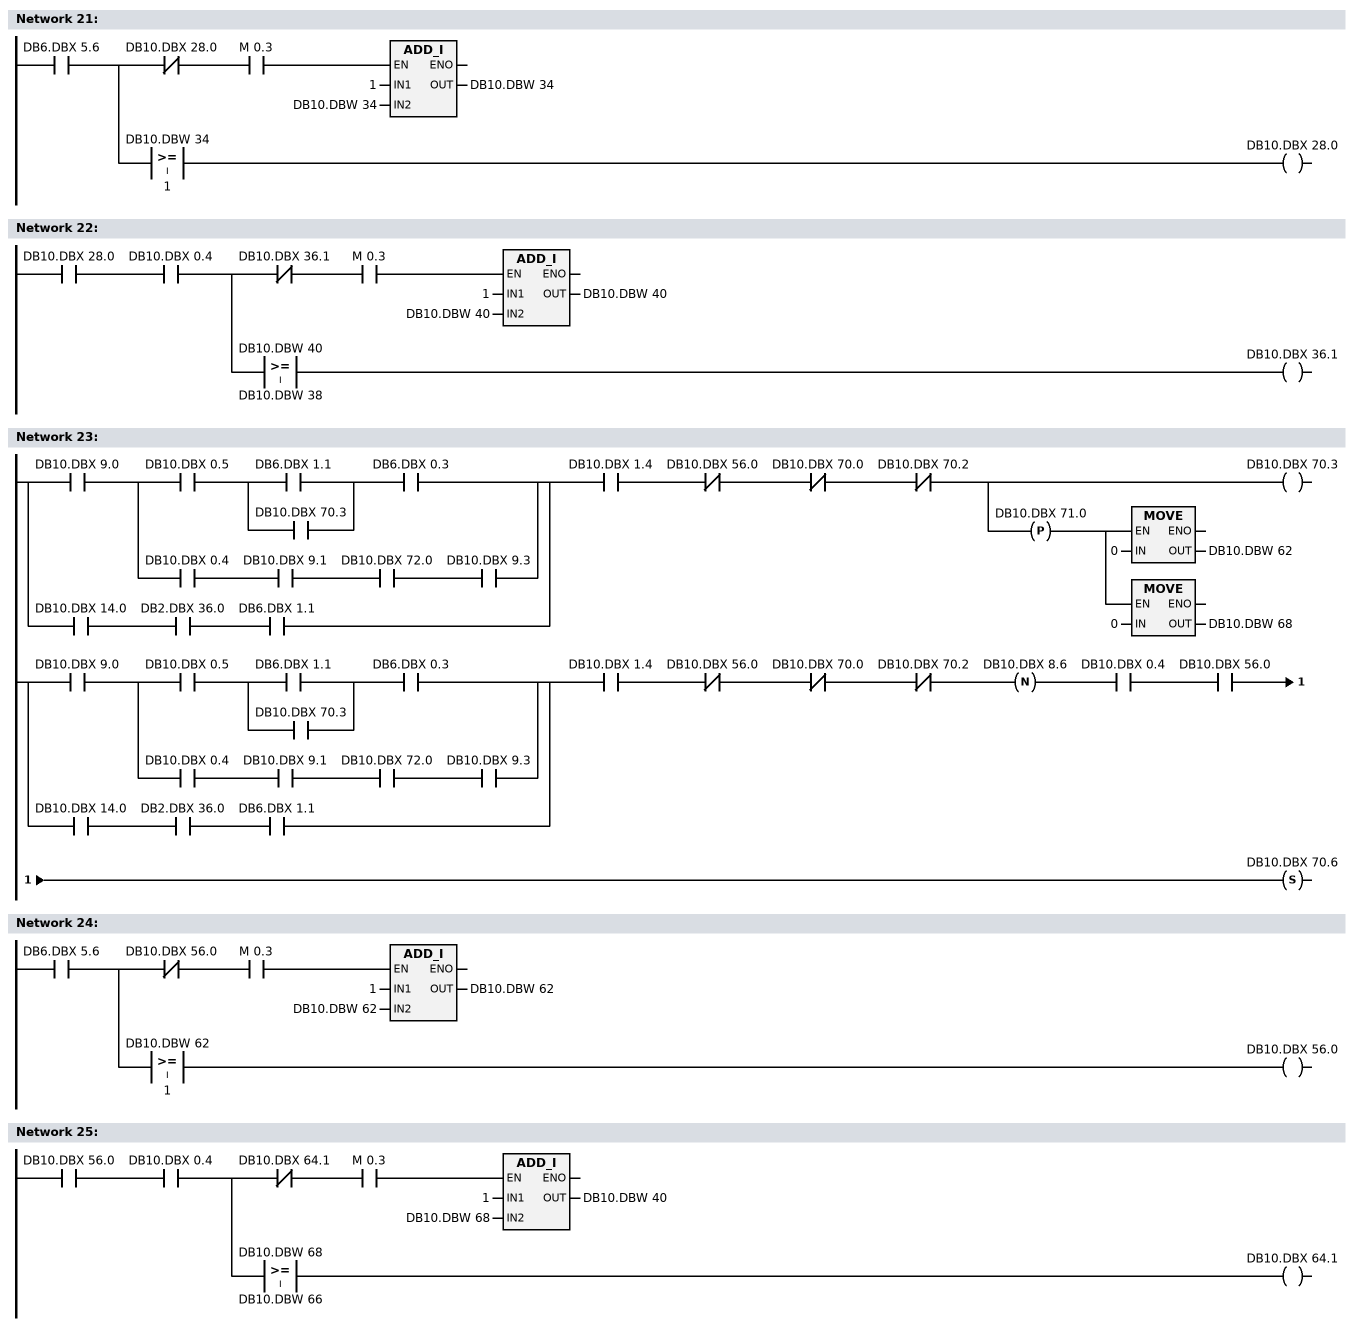
NETWORK
TITLE =
      A     DB6.DBX 5.6;
      =     L 0.0;
      A     L 0.0;
      AN    DB10.DBX 28.0;
      A     M 0.3;
      JNB   M018;
      L     1;
      L     DB10.DBW 34;
      +I;
      T     DB10.DBW 34;
M018: NOP   0;
      A     L 0.0;
      A(;
      L     DB10.DBW 34;
      L     1;
      >=I;
      );
      =     DB10.DBX 28.0;
NETWORK
TITLE =
      A     DB10.DBX 28.0;
      A     DB10.DBX 0.4;
      =     L 0.0;
      A     L 0.0;
      AN    DB10.DBX 36.1;
      A     M 0.3;
      JNB   M019;
      L     1;
      L     DB10.DBW 40;
      +I;
      T     DB10.DBW 40;
M019: NOP   0;
      A     L 0.0;
      A(;
      L     DB10.DBW 40;
      L     DB10.DBW 38;
      >=I;
      );
      =     DB10.DBX 36.1;
NETWORK
TITLE =
      A(;
      A     DB10.DBX 9.0;
      A(;
      A     DB10.DBX 0.5;
      A(;
      O     DB6.DBX 1.1;
      O     DB10.DBX 70.3;
      );
      A     DB6.DBX 0.3;
      O;
      A     DB10.DBX 0.4;
      A     DB10.DBX 9.1;
      A     DB10.DBX 72.0;
      A     DB10.DBX 9.3;
      );
      O;
      A     DB10.DBX 14.0;
      A     DB2.DBX 36.0;
      A     DB6.DBX 1.1;
      );
      A     DB10.DBX 1.4;
      AN    DB10.DBX 56.0;
      AN    DB10.DBX 70.0;
      AN    DB10.DBX 70.2;
      =     L 0.0;
      A     L 0.0;
      BLD   102;
      =     DB10.DBX 70.3;
      A(;
      A     L 0.0;
      FN    DB10.DBX 8.6;
      );
      A     DB10.DBX 0.4;
      A     DB10.DBX 56.0;
      S     DB10.DBX 70.6;
      A     L 0.0;
      FP    DB10.DBX 71.0;
      =     L 0.1;
      A     L 0.1;
      JNB   M020;
      L     0;
      T     DB10.DBW 62;
M020: NOP   0;
      A     L 0.1;
      JNB   M021;
      L     0;
      T     DB10.DBW 68;
M021: NOP   0;
NETWORK
TITLE =
      A     DB6.DBX 5.6;
      =     L 0.0;
      A     L 0.0;
      AN    DB10.DBX 56.0;
      A     M 0.3;
      JNB   M022;
      L     1;
      L     DB10.DBW 62;
      +I;
      T     DB10.DBW 62;
M022: NOP   0;
      A     L 0.0;
      A(;
      L     DB10.DBW 62;
      L     1;
      >=I;
      );
      =     DB10.DBX 56.0;
NETWORK
TITLE =
      A     DB10.DBX 56.0;
      A     DB10.DBX 0.4;
      =     L 0.0;
      A     L 0.0;
      AN    DB10.DBX 64.1;
      A     M 0.3;
      JNB   M023;
      L     1;
      L     DB10.DBW 68;
      +I;
      T     DB10.DBW 40;
M023: NOP   0;
      A     L 0.0;
      A(;
      L     DB10.DBW 68;
      L     DB10.DBW 66;
      >=I;
      );
      =     DB10.DBX 64.1;
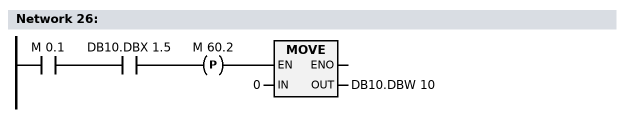
NETWORK
TITLE =
      A     M 0.1;
      A     DB10.DBX 1.5;
      FP    M 60.2;
      JNB   M024;
      L     0;
      T     DB10.DBW 10;
M024: NOP   0;
END_FUNCTION

FUNCTION FC 13 : VOID
AUTHOR : Kamillas
VERSION : 0.1
BEGIN
// (block stored without names or comments; labels and parameter names are numbered)
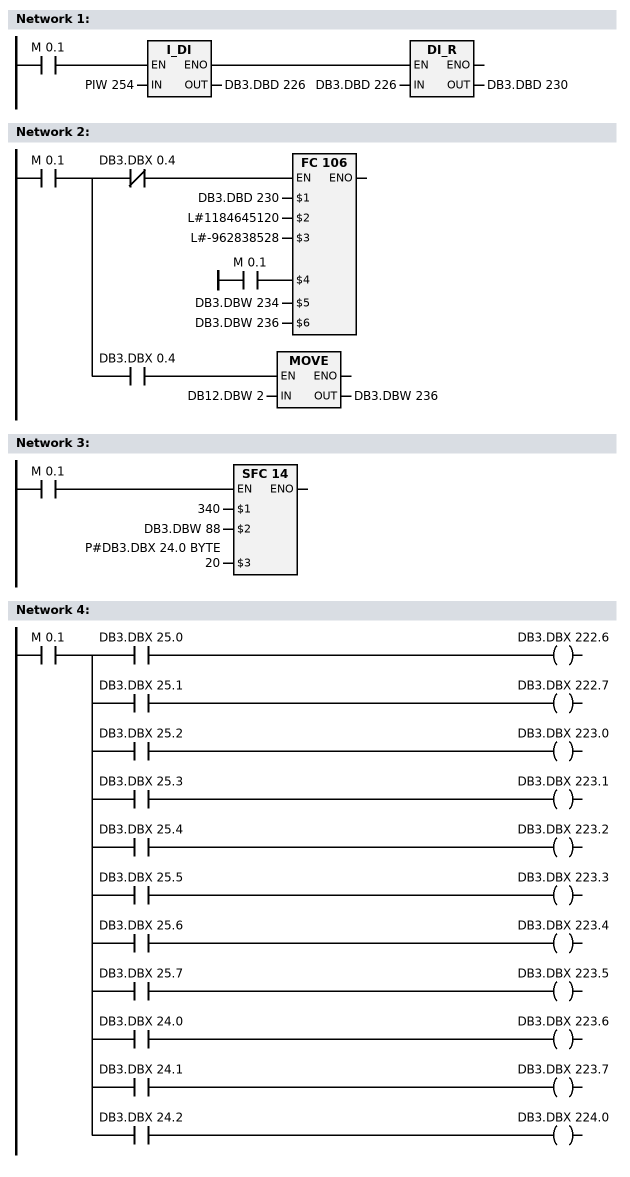
NETWORK
TITLE =
      A(;
      A     M 0.1;
      JNB   M001;
      L     PIW 254;
      ITD;
      T     DB3.DBD 226;
      SET;
      SAVE;
      CLR;
M001: A     BR;
      );
      JNB   M002;
      L     DB3.DBD 226;
      DTR;
      T     DB3.DBD 230;
M002: NOP   0;
NETWORK
TITLE =
      A     M 0.1;
      =     L 0.0;
      A     M 0.1;
      =     L 0.1;
      BLD   103;
      A     L 0.0;
      AN    DB3.DBX 0.4;
      JNB   M003;
      CALL  FC 106 (
           $1                       := DB3.DBD 230,
           $2                       := L#1184645120,
           $3                       := L#-962838528,
           $4                       := L 0.1,
           $5                       := DB3.DBW 234,
           $6                       := DB3.DBW 236);
M003: NOP   0;
      A     L 0.0;
      A     DB3.DBX 0.4;
      JNB   M004;
      L     DB12.DBW 2;
      T     DB3.DBW 236;
M004: NOP   0;
NETWORK
TITLE =
      A     M 0.1;
      JNB   M005;
      CALL  SFC 14 (
           $1                       := 340,
           $2                       := DB3.DBW 88,
           $3                       := P#DB3.DBX 24.0 BYTE 20);
M005: NOP   0;
NETWORK
TITLE =
      A     M 0.1;
      =     L 0.0;
      A     L 0.0;
      A     DB3.DBX 25.0;
      =     DB3.DBX 222.6;
      A     L 0.0;
      A     DB3.DBX 25.1;
      =     DB3.DBX 222.7;
      A     L 0.0;
      A     DB3.DBX 25.2;
      =     DB3.DBX 223.0;
      A     L 0.0;
      A     DB3.DBX 25.3;
      =     DB3.DBX 223.1;
      A     L 0.0;
      A     DB3.DBX 25.4;
      =     DB3.DBX 223.2;
      A     L 0.0;
      A     DB3.DBX 25.5;
      =     DB3.DBX 223.3;
      A     L 0.0;
      A     DB3.DBX 25.6;
      =     DB3.DBX 223.4;
      A     L 0.0;
      A     DB3.DBX 25.7;
      =     DB3.DBX 223.5;
      A     L 0.0;
      A     DB3.DBX 24.0;
      =     DB3.DBX 223.6;
      A     L 0.0;
      A     DB3.DBX 24.1;
      =     DB3.DBX 223.7;
      A     L 0.0;
      A     DB3.DBX 24.2;
      =     DB3.DBX 224.0;
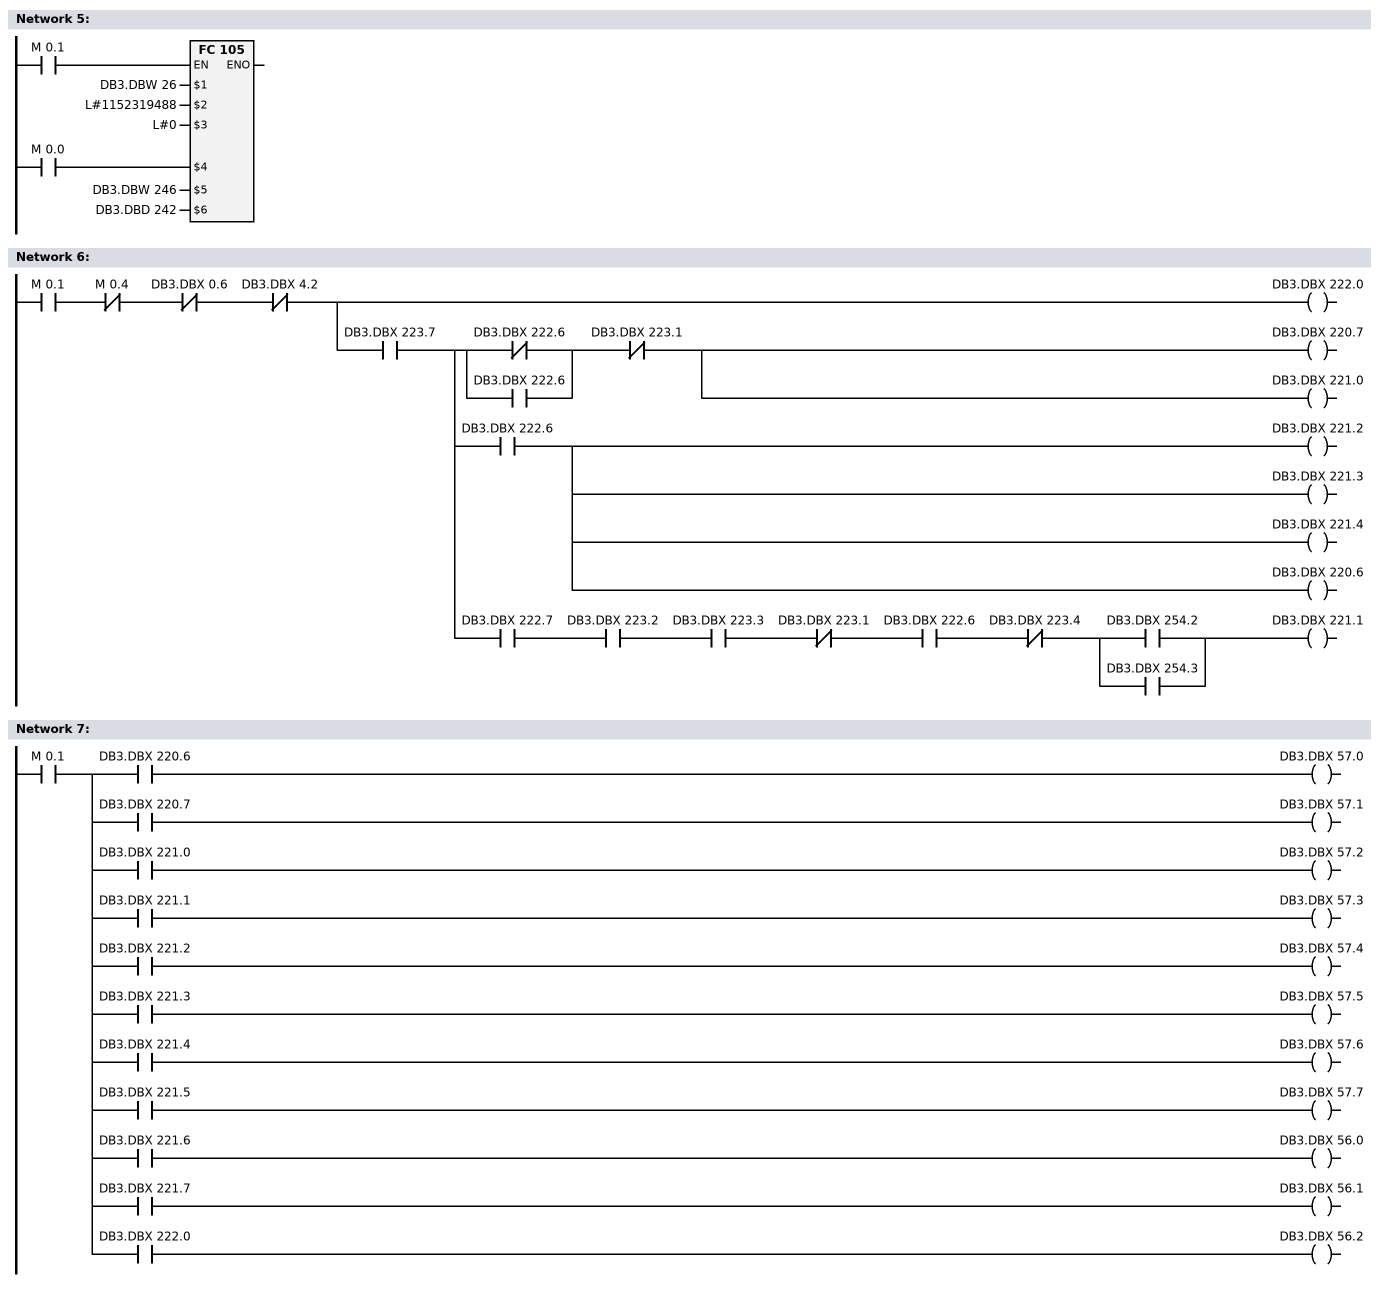
NETWORK
TITLE =
      A     M 0.0;
      =     L 0.0;
      BLD   103;
      A     M 0.1;
      JNB   M006;
      CALL  FC 105 (
           $1                       := DB3.DBW 26,
           $2                       := L#1152319488,
           $3                       := L#0,
           $4                       := L 0.0,
           $5                       := DB3.DBW 246,
           $6                       := DB3.DBD 242);
M006: NOP   0;
NETWORK
TITLE =
      A     M 0.1;
      AN    M 0.4;
      AN    DB3.DBX 0.6;
      AN    DB3.DBX 4.2;
      =     L 0.0;
      A     L 0.0;
      BLD   102;
      =     DB3.DBX 222.0;
      A     L 0.0;
      A     DB3.DBX 223.7;
      =     L 0.1;
      A     L 0.1;
      A(;
      ON    DB3.DBX 222.6;
      O     DB3.DBX 222.6;
      );
      AN    DB3.DBX 223.1;
      =     DB3.DBX 220.7;
      =     DB3.DBX 221.0;
      A     L 0.1;
      A     DB3.DBX 222.6;
      =     DB3.DBX 221.2;
      =     DB3.DBX 221.3;
      =     DB3.DBX 221.4;
      =     DB3.DBX 220.6;
      A     L 0.1;
      A     DB3.DBX 222.7;
      A     DB3.DBX 223.2;
      A     DB3.DBX 223.3;
      AN    DB3.DBX 223.1;
      A     DB3.DBX 222.6;
      AN    DB3.DBX 223.4;
      A(;
      O     DB3.DBX 254.2;
      O     DB3.DBX 254.3;
      );
      =     DB3.DBX 221.1;
NETWORK
TITLE =
      A     M 0.1;
      =     L 0.0;
      A     L 0.0;
      A     DB3.DBX 220.6;
      =     DB3.DBX 57.0;
      A     L 0.0;
      A     DB3.DBX 220.7;
      =     DB3.DBX 57.1;
      A     L 0.0;
      A     DB3.DBX 221.0;
      =     DB3.DBX 57.2;
      A     L 0.0;
      A     DB3.DBX 221.1;
      =     DB3.DBX 57.3;
      A     L 0.0;
      A     DB3.DBX 221.2;
      =     DB3.DBX 57.4;
      A     L 0.0;
      A     DB3.DBX 221.3;
      =     DB3.DBX 57.5;
      A     L 0.0;
      A     DB3.DBX 221.4;
      =     DB3.DBX 57.6;
      A     L 0.0;
      A     DB3.DBX 221.5;
      =     DB3.DBX 57.7;
      A     L 0.0;
      A     DB3.DBX 221.6;
      =     DB3.DBX 56.0;
      A     L 0.0;
      A     DB3.DBX 221.7;
      =     DB3.DBX 56.1;
      A     L 0.0;
      A     DB3.DBX 222.0;
      =     DB3.DBX 56.2;
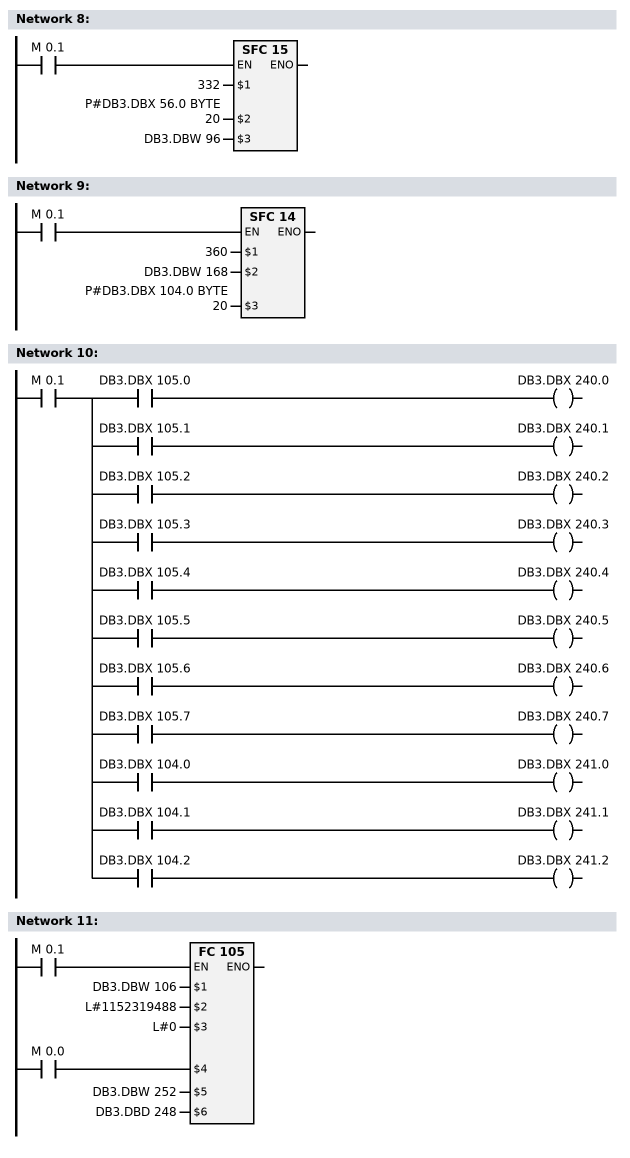
NETWORK
TITLE =
      A     M 0.1;
      JNB   M007;
      CALL  SFC 15 (
           $1                       := 332,
           $2                       := P#DB3.DBX 56.0 BYTE 20,
           $3                       := DB3.DBW 96);
M007: NOP   0;
NETWORK
TITLE =
      A     M 0.1;
      JNB   M008;
      CALL  SFC 14 (
           $1                       := 360,
           $2                       := DB3.DBW 168,
           $3                       := P#DB3.DBX 104.0 BYTE 20);
M008: NOP   0;
NETWORK
TITLE =
      A     M 0.1;
      =     L 0.0;
      A     L 0.0;
      A     DB3.DBX 105.0;
      =     DB3.DBX 240.0;
      A     L 0.0;
      A     DB3.DBX 105.1;
      =     DB3.DBX 240.1;
      A     L 0.0;
      A     DB3.DBX 105.2;
      =     DB3.DBX 240.2;
      A     L 0.0;
      A     DB3.DBX 105.3;
      =     DB3.DBX 240.3;
      A     L 0.0;
      A     DB3.DBX 105.4;
      =     DB3.DBX 240.4;
      A     L 0.0;
      A     DB3.DBX 105.5;
      =     DB3.DBX 240.5;
      A     L 0.0;
      A     DB3.DBX 105.6;
      =     DB3.DBX 240.6;
      A     L 0.0;
      A     DB3.DBX 105.7;
      =     DB3.DBX 240.7;
      A     L 0.0;
      A     DB3.DBX 104.0;
      =     DB3.DBX 241.0;
      A     L 0.0;
      A     DB3.DBX 104.1;
      =     DB3.DBX 241.1;
      A     L 0.0;
      A     DB3.DBX 104.2;
      =     DB3.DBX 241.2;
NETWORK
TITLE =
      A     M 0.0;
      =     L 0.0;
      BLD   103;
      A     M 0.1;
      JNB   M009;
      CALL  FC 105 (
           $1                       := DB3.DBW 106,
           $2                       := L#1152319488,
           $3                       := L#0,
           $4                       := L 0.0,
           $5                       := DB3.DBW 252,
           $6                       := DB3.DBD 248);
M009: NOP   0;
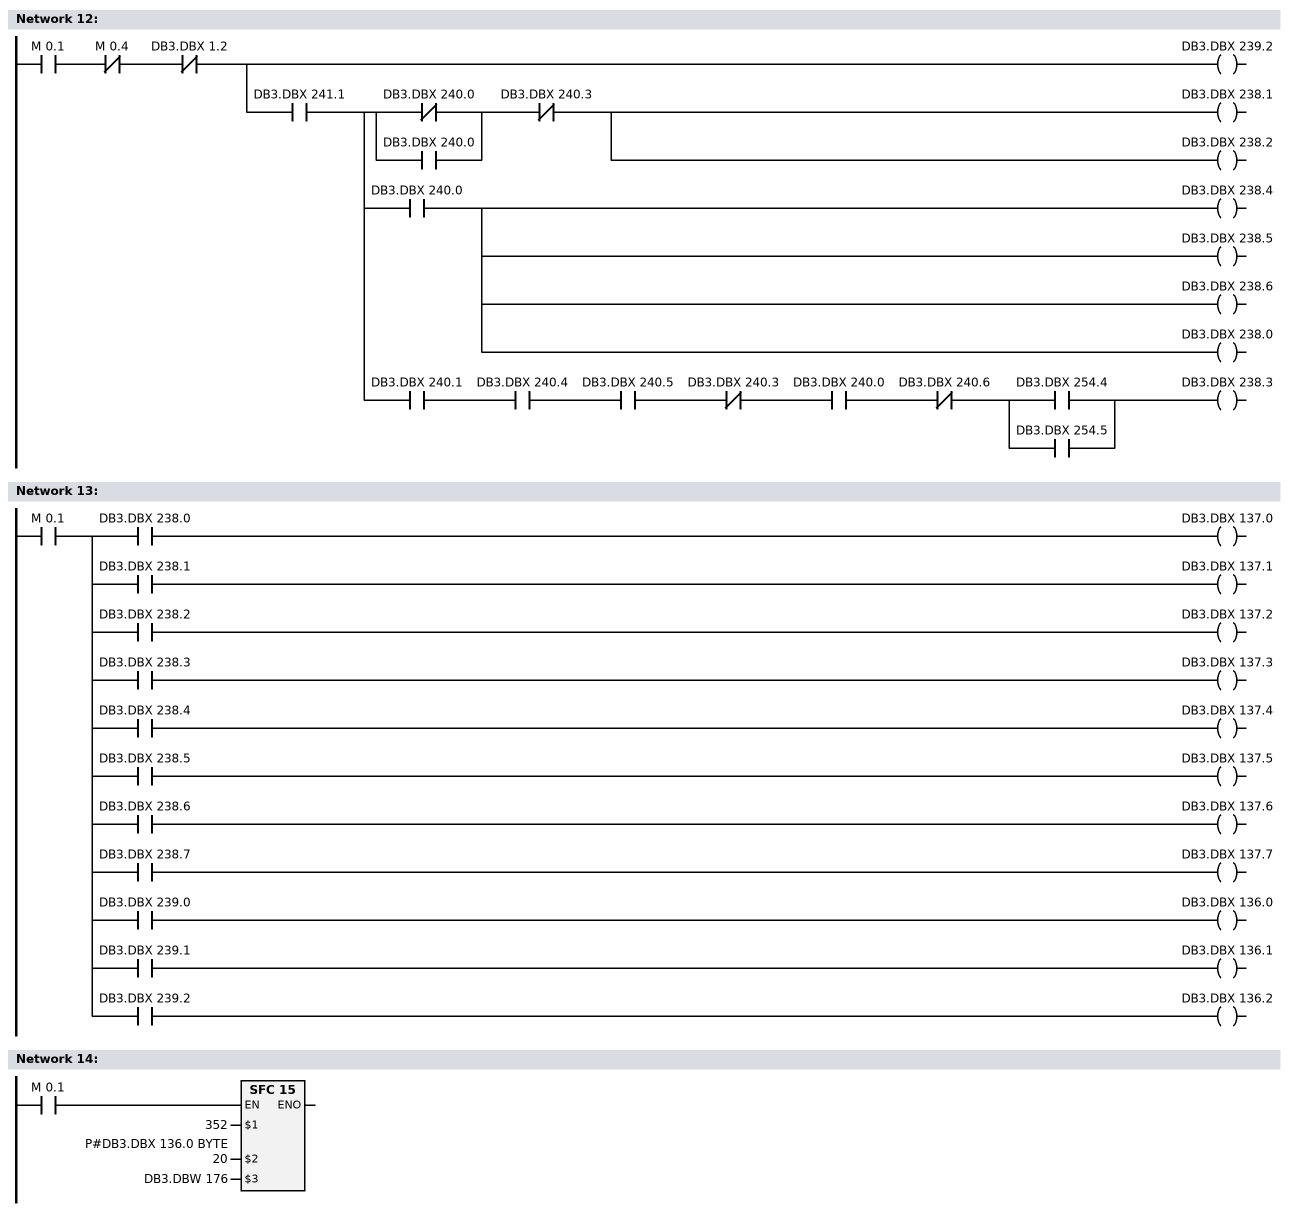
NETWORK
TITLE =
      A     M 0.1;
      AN    M 0.4;
      AN    DB3.DBX 1.2;
      =     L 0.0;
      A     L 0.0;
      BLD   102;
      =     DB3.DBX 239.2;
      A     L 0.0;
      A     DB3.DBX 241.1;
      =     L 0.1;
      A     L 0.1;
      A(;
      ON    DB3.DBX 240.0;
      O     DB3.DBX 240.0;
      );
      AN    DB3.DBX 240.3;
      =     DB3.DBX 238.1;
      =     DB3.DBX 238.2;
      A     L 0.1;
      A     DB3.DBX 240.0;
      =     DB3.DBX 238.4;
      =     DB3.DBX 238.5;
      =     DB3.DBX 238.6;
      =     DB3.DBX 238.0;
      A     L 0.1;
      A     DB3.DBX 240.1;
      A     DB3.DBX 240.4;
      A     DB3.DBX 240.5;
      AN    DB3.DBX 240.3;
      A     DB3.DBX 240.0;
      AN    DB3.DBX 240.6;
      A(;
      O     DB3.DBX 254.4;
      O     DB3.DBX 254.5;
      );
      =     DB3.DBX 238.3;
NETWORK
TITLE =
      A     M 0.1;
      =     L 0.0;
      A     L 0.0;
      A     DB3.DBX 238.0;
      =     DB3.DBX 137.0;
      A     L 0.0;
      A     DB3.DBX 238.1;
      =     DB3.DBX 137.1;
      A     L 0.0;
      A     DB3.DBX 238.2;
      =     DB3.DBX 137.2;
      A     L 0.0;
      A     DB3.DBX 238.3;
      =     DB3.DBX 137.3;
      A     L 0.0;
      A     DB3.DBX 238.4;
      =     DB3.DBX 137.4;
      A     L 0.0;
      A     DB3.DBX 238.5;
      =     DB3.DBX 137.5;
      A     L 0.0;
      A     DB3.DBX 238.6;
      =     DB3.DBX 137.6;
      A     L 0.0;
      A     DB3.DBX 238.7;
      =     DB3.DBX 137.7;
      A     L 0.0;
      A     DB3.DBX 239.0;
      =     DB3.DBX 136.0;
      A     L 0.0;
      A     DB3.DBX 239.1;
      =     DB3.DBX 136.1;
      A     L 0.0;
      A     DB3.DBX 239.2;
      =     DB3.DBX 136.2;
NETWORK
TITLE =
      A     M 0.1;
      JNB   M010;
      CALL  SFC 15 (
           $1                       := 352,
           $2                       := P#DB3.DBX 136.0 BYTE 20,
           $3                       := DB3.DBW 176);
M010: NOP   0;
END_FUNCTION

FUNCTION FC 14 : VOID
VERSION : 0.1
BEGIN
// (block stored without names or comments; labels and parameter names are numbered)
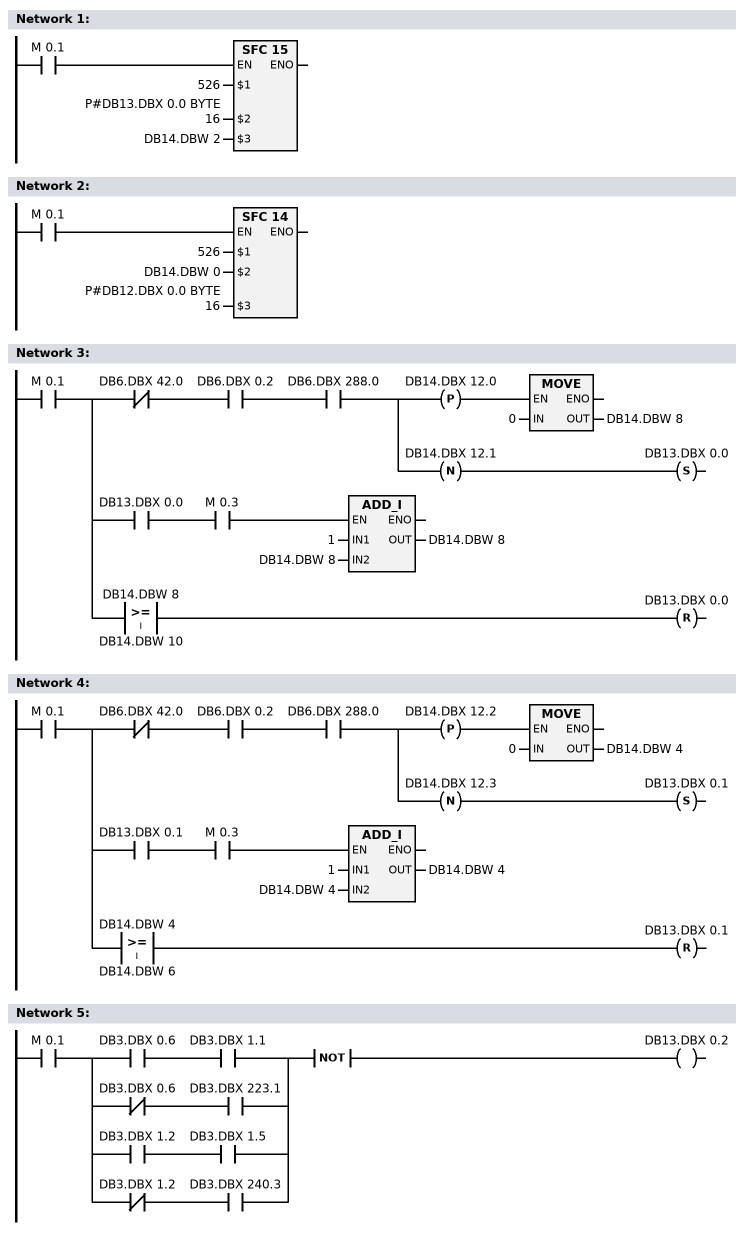
NETWORK
TITLE =
      A     M 0.1;
      JNB   M001;
      CALL  SFC 15 (
           $1                       := 526,
           $2                       := P#DB13.DBX 0.0 BYTE 16,
           $3                       := DB14.DBW 2);
M001: NOP   0;
NETWORK
TITLE =
      A     M 0.1;
      JNB   M002;
      CALL  SFC 14 (
           $1                       := 526,
           $2                       := DB14.DBW 0,
           $3                       := P#DB12.DBX 0.0 BYTE 16);
M002: NOP   0;
NETWORK
TITLE =
      A     M 0.1;
      =     L 0.0;
      A     L 0.0;
      AN    DB6.DBX 42.0;
      A     DB6.DBX 0.2;
      A     DB6.DBX 288.0;
      =     L 0.1;
      A     L 0.1;
      FP    DB14.DBX 12.0;
      JNB   M003;
      L     0;
      T     DB14.DBW 8;
M003: NOP   0;
      A     L 0.1;
      FN    DB14.DBX 12.1;
      S     DB13.DBX 0.0;
      A     L 0.0;
      A     DB13.DBX 0.0;
      A     M 0.3;
      JNB   M004;
      L     1;
      L     DB14.DBW 8;
      +I;
      T     DB14.DBW 8;
M004: NOP   0;
      A     L 0.0;
      A(;
      L     DB14.DBW 8;
      L     DB14.DBW 10;
      >=I;
      );
      R     DB13.DBX 0.0;
NETWORK
TITLE =
      A     M 0.1;
      =     L 0.0;
      A     L 0.0;
      AN    DB6.DBX 42.0;
      A     DB6.DBX 0.2;
      A     DB6.DBX 288.0;
      =     L 0.1;
      A     L 0.1;
      FP    DB14.DBX 12.2;
      JNB   M005;
      L     0;
      T     DB14.DBW 4;
M005: NOP   0;
      A     L 0.1;
      FN    DB14.DBX 12.3;
      S     DB13.DBX 0.1;
      A     L 0.0;
      A     DB13.DBX 0.1;
      A     M 0.3;
      JNB   M006;
      L     1;
      L     DB14.DBW 4;
      +I;
      T     DB14.DBW 4;
M006: NOP   0;
      A     L 0.0;
      A(;
      L     DB14.DBW 4;
      L     DB14.DBW 6;
      >=I;
      );
      R     DB13.DBX 0.1;
NETWORK
TITLE =
      A     M 0.1;
      A(;
      A     DB3.DBX 0.6;
      A     DB3.DBX 1.1;
      O;
      AN    DB3.DBX 0.6;
      A     DB3.DBX 223.1;
      O;
      A     DB3.DBX 1.2;
      A     DB3.DBX 1.5;
      O;
      AN    DB3.DBX 1.2;
      A     DB3.DBX 240.3;
      );
      NOT;
      =     DB13.DBX 0.2;
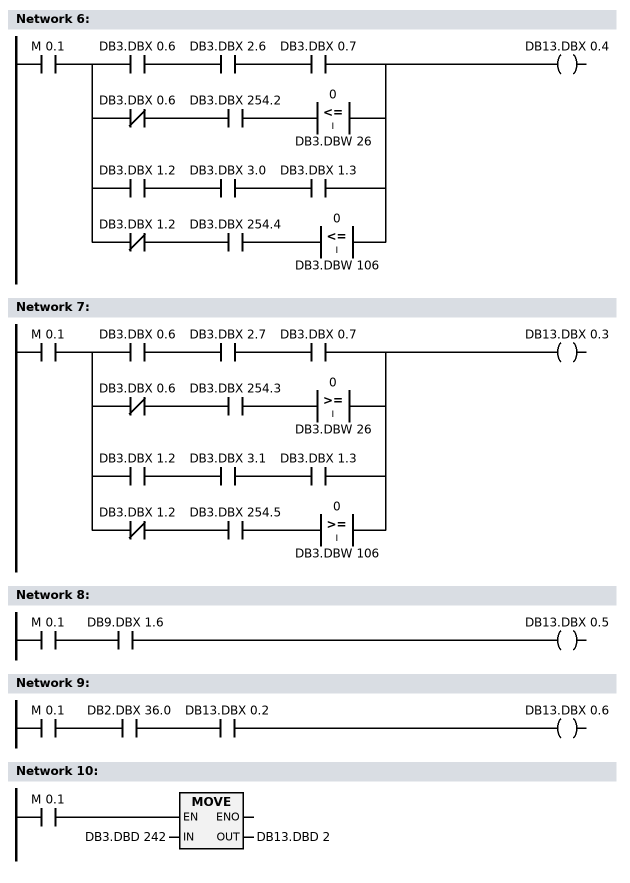
NETWORK
TITLE =
      A     M 0.1;
      A(;
      A     DB3.DBX 0.6;
      A     DB3.DBX 2.6;
      A     DB3.DBX 0.7;
      O;
      AN    DB3.DBX 0.6;
      A     DB3.DBX 254.2;
      A(;
      L     0;
      L     DB3.DBW 26;
      <=I;
      );
      O;
      A     DB3.DBX 1.2;
      A     DB3.DBX 3.0;
      A     DB3.DBX 1.3;
      O;
      AN    DB3.DBX 1.2;
      A     DB3.DBX 254.4;
      A(;
      L     0;
      L     DB3.DBW 106;
      <=I;
      );
      );
      =     DB13.DBX 0.4;
NETWORK
TITLE =
      A     M 0.1;
      A(;
      A     DB3.DBX 0.6;
      A     DB3.DBX 2.7;
      A     DB3.DBX 0.7;
      O;
      AN    DB3.DBX 0.6;
      A     DB3.DBX 254.3;
      A(;
      L     0;
      L     DB3.DBW 26;
      >=I;
      );
      O;
      A     DB3.DBX 1.2;
      A     DB3.DBX 3.1;
      A     DB3.DBX 1.3;
      O;
      AN    DB3.DBX 1.2;
      A     DB3.DBX 254.5;
      A(;
      L     0;
      L     DB3.DBW 106;
      >=I;
      );
      );
      =     DB13.DBX 0.3;
NETWORK
TITLE =
      A     M 0.1;
      A     DB9.DBX 1.6;
      =     DB13.DBX 0.5;
NETWORK
TITLE =
      A     M 0.1;
      A     DB2.DBX 36.0;
      A     DB13.DBX 0.2;
      =     DB13.DBX 0.6;
NETWORK
TITLE =
      A     M 0.1;
      JNB   M007;
      L     DB3.DBD 242;
      T     DB13.DBD 2;
M007: NOP   0;
END_FUNCTION

// FC 105: know-how protected block, not included

// FC 106: know-how protected block, not included

DATA_BLOCK DB 1
AUTHOR : Kamillas
VERSION : 0.1
BEGIN
// 14 bytes; values not shown
END_DATA_BLOCK

DATA_BLOCK DB 2
AUTHOR : Kamillas
VERSION : 0.1
BEGIN
// 38 bytes; values not shown
END_DATA_BLOCK

DATA_BLOCK DB 3
AUTHOR : Kamillas
VERSION : 0.1
BEGIN
// 256 bytes; values not shown
END_DATA_BLOCK

DATA_BLOCK DB 4
AUTHOR : Kamillas
VERSION : 0.1
BEGIN
// 8 bytes; values not shown
END_DATA_BLOCK

DATA_BLOCK DB 5
AUTHOR : Kamillas
VERSION : 0.1
BEGIN
// 120 bytes; values not shown
END_DATA_BLOCK

DATA_BLOCK DB 6
AUTHOR : Kamillas
VERSION : 0.1
BEGIN
// 360 bytes; values not shown
END_DATA_BLOCK

DATA_BLOCK DB 7
AUTHOR : Kamillas
VERSION : 0.1
BEGIN
// 24 bytes; values not shown
END_DATA_BLOCK

DATA_BLOCK DB 8
AUTHOR : Kamillas
VERSION : 0.1
BEGIN
// 62 bytes; values not shown
END_DATA_BLOCK

DATA_BLOCK DB 9
AUTHOR : Kamillas
VERSION : 0.1
BEGIN
// 24 bytes; values not shown
END_DATA_BLOCK

DATA_BLOCK DB 10
AUTHOR : Kamillas
VERSION : 0.1
BEGIN
// 74 bytes; values not shown
END_DATA_BLOCK

DATA_BLOCK DB 11
AUTHOR : Kamilas
VERSION : 0.1
BEGIN
// 32 bytes; values not shown
END_DATA_BLOCK

DATA_BLOCK DB 12
VERSION : 0.1
BEGIN
// 18 bytes; values not shown
END_DATA_BLOCK

DATA_BLOCK DB 13
VERSION : 0.1
BEGIN
// 18 bytes; values not shown
END_DATA_BLOCK

DATA_BLOCK DB 14
VERSION : 0.1
BEGIN
// 14 bytes; values not shown
END_DATA_BLOCK

ORGANIZATION_BLOCK OB 1
AUTHOR : Kamillas
VERSION : 0.1
BEGIN
// (block stored without names or comments; labels and parameter names are numbered)
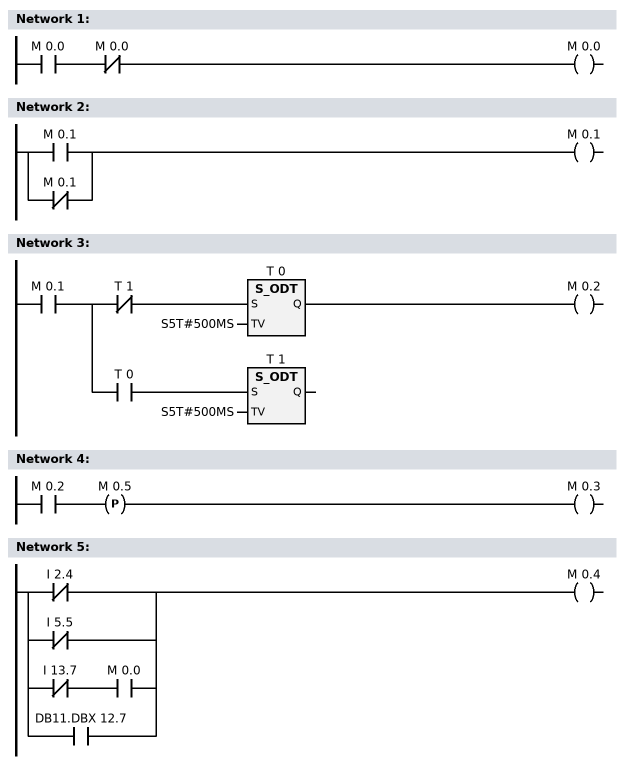
NETWORK
TITLE =
      A     M 0.0;
      AN    M 0.0;
      =     M 0.0;
NETWORK
TITLE =
      O     M 0.1;
      ON    M 0.1;
      =     M 0.1;
NETWORK
TITLE =
      A     M 0.1;
      =     L 20.0;
      A     L 20.0;
      AN    T 1;
      L     S5T#500MS;
      SD    T 0;
      NOP   0;
      NOP   0;
      NOP   0;
      A     T 0;
      =     M 0.2;
      A     L 20.0;
      A     T 0;
      L     S5T#500MS;
      SD    T 1;
      NOP   0;
      NOP   0;
      NOP   0;
      NOP   0;
NETWORK
TITLE =
      A     M 0.2;
      FP    M 0.5;
      =     M 0.3;
NETWORK
TITLE =
      ON    I 2.4;
      ON    I 5.5;
      O;
      AN    I 13.7;
      A     M 0.0;
      O     DB11.DBX 12.7;
      =     M 0.4;
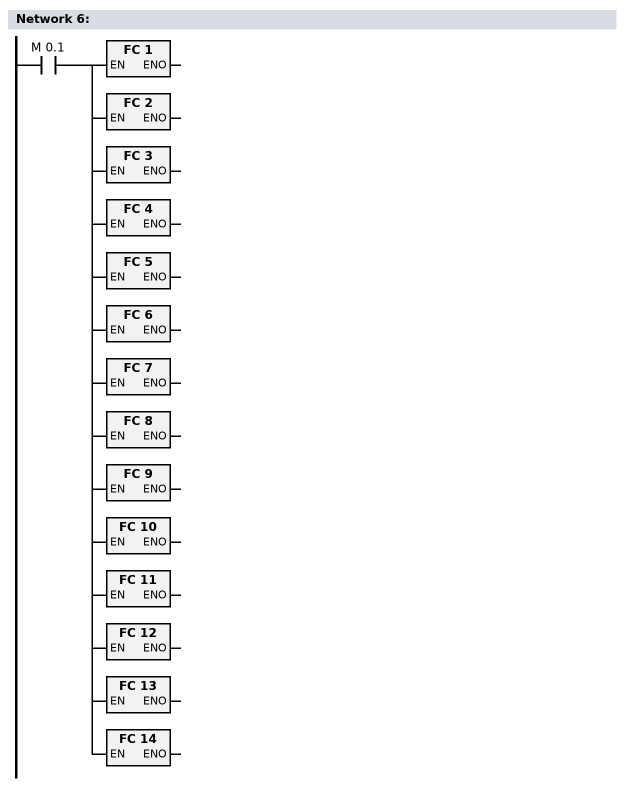
NETWORK
TITLE =
      A     M 0.1;
      =     L 20.0;
      A     L 20.0;
      JNB   M001;
      CALL  FC 1;
M001: NOP   0;
      A     L 20.0;
      JNB   M002;
      CALL  FC 2;
M002: NOP   0;
      A     L 20.0;
      JNB   M003;
      CALL  FC 3;
M003: NOP   0;
      A     L 20.0;
      JNB   M004;
      CALL  FC 4;
M004: NOP   0;
      A     L 20.0;
      JNB   M005;
      CALL  FC 5;
M005: NOP   0;
      A     L 20.0;
      JNB   M006;
      CALL  FC 6;
M006: NOP   0;
      A     L 20.0;
      JNB   M007;
      CALL  FC 7;
M007: NOP   0;
      A     L 20.0;
      JNB   M008;
      CALL  FC 8;
M008: NOP   0;
      A     L 20.0;
      JNB   M009;
      CALL  FC 9;
M009: NOP   0;
      A     L 20.0;
      JNB   M010;
      CALL  FC 10;
M010: NOP   0;
      A     L 20.0;
      JNB   M011;
      CALL  FC 11;
M011: NOP   0;
      A     L 20.0;
      JNB   M012;
      CALL  FC 12;
M012: NOP   0;
      A     L 20.0;
      JNB   M013;
      CALL  FC 13;
M013: NOP   0;
      A     L 20.0;
      JNB   M014;
      CALL  FC 14;
M014: NOP   0;
END_ORGANIZATION_BLOCK

ORGANIZATION_BLOCK OB 82
AUTHOR : Kamillas
VERSION : 0.1
BEGIN
// (block stored without names or comments; labels and parameter names are numbered)
END_ORGANIZATION_BLOCK

ORGANIZATION_BLOCK OB 86
AUTHOR : Kamillas
VERSION : 0.1
BEGIN
// (block stored without names or comments; labels and parameter names are numbered)
END_ORGANIZATION_BLOCK

ORGANIZATION_BLOCK OB 121
AUTHOR : Kamillas
VERSION : 0.1
BEGIN
// (block stored without names or comments; labels and parameter names are numbered)
END_ORGANIZATION_BLOCK

ORGANIZATION_BLOCK OB 122
AUTHOR : Kamillas
VERSION : 0.1
BEGIN
// (block stored without names or comments; labels and parameter names are numbered)
END_ORGANIZATION_BLOCK
